C07310=1226.030,289.188,-65.591,-176.498,6.719,148.208
C07311=1226.024,289.461,-65.622,-176.496,6.721,148.208
C07312=1226.020,289.735,-65.655,-176.493,6.724,148.208
C07313=1226.015,290.009,-65.686,-176.491,6.726,148.208
C07314=1226.010,290.258,-65.715,-176.488,6.729,148.208
C07315=1226.006,290.505,-65.743,-176.486,6.731,148.208
C07316=1226.002,290.754,-65.772,-176.483,6.733,148.207
C07317=1225.998,291.003,-65.802,-176.481,6.735,148.207
C07318=1225.994,291.251,-65.830,-176.478,6.738,148.207
C07319=1225.989,291.499,-65.859,-176.476,6.741,148.207
C07320=1225.985,291.748,-65.888,-176.474,6.742,148.207
C07321=1225.980,291.996,-65.917,-176.471,6.746,148.207
C07322=1225.975,292.244,-65.945,-176.469,6.748,148.207
C07323=1225.972,292.492,-65.974,-176.467,6.750,148.207
C07324=1225.967,292.741,-66.003,-176.464,6.752,148.206
C07325=1225.963,292.989,-66.032,-176.462,6.755,148.206
C07326=1225.958,293.237,-66.061,-176.459,6.757,148.206
C07327=1225.954,293.486,-66.090,-176.457,6.759,148.206
C07328=1225.951,293.734,-66.119,-176.455,6.761,148.206
C07329=1225.945,293.982,-66.148,-176.452,6.764,148.206
C07330=1225.941,294.230,-66.177,-176.450,6.767,148.206
C07331=1225.937,294.478,-66.206,-176.448,6.769,148.206
C07332=1225.933,294.727,-66.235,-176.445,6.771,148.206
C07333=1225.928,294.975,-66.265,-176.443,6.774,148.206
C07334=1225.924,295.223,-66.292,-176.440,6.776,148.206
C07335=1225.920,295.472,-66.322,-176.438,6.778,148.206
C07336=1225.916,295.720,-66.351,-176.435,6.781,148.205
C07337=1225.912,295.968,-66.381,-176.433,6.783,148.205
C07338=1225.906,296.216,-66.409,-176.431,6.785,148.205
C07339=1225.902,296.465,-66.439,-176.428,6.788,148.205
C07340=1225.898,296.713,-66.468,-176.426,6.791,148.205
C07341=1225.894,296.962,-66.497,-176.424,6.792,148.205
C07342=1225.889,297.210,-66.526,-176.422,6.795,148.205
C07343=1225.885,297.458,-66.555,-176.419,6.798,148.205
C07344=1225.881,297.706,-66.584,-176.417,6.800,148.205
C07345=1225.877,297.954,-66.614,-176.415,6.802,148.205
C07346=1225.873,298.203,-66.642,-176.412,6.805,148.205
C07347=1225.868,298.451,-66.672,-176.409,6.807,148.204
C07348=1225.864,298.699,-66.701,-176.407,6.809,148.204
C07349=1225.859,298.947,-66.730,-176.405,6.812,148.204
C07350=1225.855,299.195,-66.760,-176.403,6.815,148.204
C07351=1225.851,299.443,-66.789,-176.400,6.817,148.204
C07352=1225.847,299.692,-66.818,-176.398,6.819,148.204
C07353=1225.842,299.941,-66.847,-176.395,6.822,148.204
C07354=1225.838,300.189,-66.877,-176.393,6.824,148.204
C07355=1225.833,300.436,-66.906,-176.391,6.826,148.204
C07356=1225.829,300.685,-66.935,-176.388,6.829,148.204
C07357=1225.825,300.933,-66.965,-176.386,6.831,148.204
C07358=1225.821,301.181,-66.994,-176.384,6.834,148.204
C07359=1225.817,301.429,-67.024,-176.381,6.837,148.204
C07360=1225.812,301.678,-67.054,-176.379,6.839,148.204
C07361=1225.808,301.926,-67.083,-176.377,6.841,148.203
C07362=1225.803,302.175,-67.113,-176.374,6.844,148.203
C07363=1225.799,302.422,-67.142,-176.372,6.846,148.203
C07364=1225.794,302.670,-67.171,-176.370,6.848,148.203
C07365=1225.790,302.919,-67.201,-176.367,6.851,148.203
C07366=1225.786,303.167,-67.230,-176.365,6.854,148.203
C07367=1225.782,303.415,-67.260,-176.363,6.856,148.203
C07368=1225.778,303.663,-67.289,-176.361,6.858,148.203
C07369=1225.774,303.912,-67.319,-176.358,6.861,148.203
C07370=1225.769,304.160,-67.349,-176.356,6.863,148.203
C07371=1225.764,304.409,-67.378,-176.354,6.866,148.203
C07372=1225.760,304.657,-67.408,-176.351,6.868,148.203
C07373=1225.756,304.905,-67.437,-176.349,6.871,148.203
C07374=1225.752,305.153,-67.466,-176.347,6.873,148.203
C07375=1225.748,305.401,-67.497,-176.344,6.876,148.203
C07376=1225.742,305.649,-67.526,-176.342,6.878,148.202
C07377=1225.738,305.897,-67.556,-176.340,6.880,148.202
C07378=1225.734,306.145,-67.585,-176.337,6.883,148.202
C07379=1225.730,306.394,-67.615,-176.335,6.885,148.202
C07380=1225.726,306.642,-67.644,-176.333,6.888,148.202
C07381=1225.721,306.890,-67.675,-176.330,6.891,148.202
C07382=1225.717,307.138,-67.704,-176.328,6.893,148.202
C07383=1225.713,307.386,-67.734,-176.326,6.895,148.202
C07384=1225.709,307.635,-67.763,-176.323,6.898,148.202
C07385=1225.704,307.883,-67.794,-176.321,6.900,148.202
C07386=1225.700,308.131,-67.823,-176.319,6.903,148.202
C07387=1225.696,308.379,-67.853,-176.316,6.906,148.202
C07388=1225.691,308.627,-67.882,-176.314,6.908,148.202
C07389=1225.687,308.875,-67.913,-176.312,6.910,148.202
C07390=1225.683,309.124,-67.943,-176.310,6.913,148.202
C07391=1225.678,309.372,-67.972,-176.307,6.915,148.202
C07392=1225.674,309.620,-68.003,-176.305,6.918,148.202
C07393=1225.670,309.868,-68.032,-176.303,6.921,148.202
C07394=1225.665,310.116,-68.062,-176.301,6.923,148.202
C07395=1225.661,310.364,-68.092,-176.298,6.925,148.202
C07396=1225.657,310.613,-68.122,-176.296,6.928,148.202
C07397=1225.653,310.861,-68.151,-176.294,6.930,148.202
C07398=1225.648,311.109,-68.182,-176.292,6.933,148.202
C07399=1225.644,311.358,-68.212,-176.289,6.936,148.202
C07400=1225.640,311.605,-68.242,-176.287,6.938,148.202
C07401=1225.636,311.854,-68.272,-176.285,6.940,148.202
C07402=1225.631,312.102,-68.302,-176.283,6.944,148.202
C07403=1225.627,312.350,-68.332,-176.280,6.946,148.202
C07404=1225.623,312.599,-68.362,-176.278,6.948,148.202
C07405=1225.619,312.846,-68.392,-176.276,6.951,148.202
C07406=1225.614,313.095,-68.422,-176.274,6.953,148.202
C07407=1225.610,313.342,-68.452,-176.271,6.956,148.202
C07408=1225.606,313.591,-68.482,-176.269,6.958,148.202
C07409=1225.601,313.839,-68.512,-176.267,6.961,148.202
C07410=1225.597,314.087,-68.542,-176.264,6.964,148.202
C07411=1225.592,314.335,-68.573,-176.262,6.966,148.202
C07412=1225.589,314.583,-68.603,-176.260,6.969,148.202
C07413=1225.584,314.832,-68.633,-176.258,6.972,148.202
C07414=1225.579,315.107,-68.667,-176.256,6.974,148.202
C07415=1225.574,315.383,-68.700,-176.253,6.977,148.202
C07416=1225.570,315.658,-68.734,-176.250,6.980,148.202
C07417=1225.565,315.935,-68.767,-176.248,6.982,148.202
C07418=1225.561,316.183,-68.798,-176.246,6.985,148.202
C07419=1225.556,316.431,-68.828,-176.243,6.987,148.202
C07420=1225.553,316.679,-68.858,-176.241,6.991,148.202
C07421=1225.548,316.927,-68.889,-176.239,6.993,148.202
C07422=1225.544,317.176,-68.918,-176.237,6.995,148.202
C07423=1225.540,317.424,-68.949,-176.234,6.998,148.202
C07424=1225.536,317.671,-68.979,-176.232,7.000,148.202
C07425=1225.531,317.920,-69.009,-176.230,7.003,148.202
C07426=1225.526,318.168,-69.040,-176.228,7.006,148.202
C07427=1225.522,318.415,-69.070,-176.226,7.008,148.202
C07428=1225.518,318.664,-69.101,-176.224,7.011,148.202
C07429=1225.514,318.912,-69.131,-176.221,7.014,148.202
C07430=1225.510,319.160,-69.162,-176.219,7.016,148.202
C07431=1225.506,319.408,-69.192,-176.217,7.018,148.202
C07432=1225.501,319.656,-69.223,-176.215,7.021,148.202
C07433=1225.497,319.905,-69.254,-176.213,7.024,148.202
C07434=1225.493,320.153,-69.283,-176.211,7.026,148.202
C07435=1225.488,320.401,-69.314,-176.208,7.029,148.202
C07436=1225.485,320.648,-69.344,-176.206,7.031,148.202
C07437=1225.480,320.896,-69.375,-176.204,7.034,148.202
C07438=1225.476,321.145,-69.406,-176.201,7.037,148.202
C07439=1225.472,321.393,-69.436,-176.200,7.039,148.202
C07440=1225.467,321.641,-69.466,-176.197,7.042,148.202
C07441=1225.462,321.889,-69.497,-176.195,7.044,148.202
C07442=1225.459,322.138,-69.527,-176.193,7.047,148.202
C07443=1225.455,322.386,-69.558,-176.191,7.050,148.202
C07444=1225.450,322.634,-69.589,-176.189,7.052,148.202
C07445=1225.446,322.881,-69.619,-176.187,7.055,148.202
C07446=1225.442,323.130,-69.650,-176.184,7.058,148.202
C07447=1225.437,323.378,-69.681,-176.182,7.060,148.202
C07448=1225.434,323.625,-69.711,-176.180,7.062,148.202
C07449=1225.430,323.874,-69.742,-176.178,7.066,148.202
C07450=1225.425,324.122,-69.773,-176.176,7.068,148.202
C07451=1225.420,324.370,-69.804,-176.173,7.071,148.202
C07452=1225.416,324.618,-69.834,-176.172,7.073,148.203
C07453=1225.412,324.866,-69.865,-176.170,7.076,148.202
C07454=1225.408,325.114,-69.896,-176.167,7.079,148.203
C07455=1225.403,325.362,-69.927,-176.165,7.081,148.203
C07456=1225.400,325.611,-69.957,-176.163,7.084,148.203
C07457=1225.395,325.859,-69.988,-176.160,7.087,148.203
C07458=1225.391,326.107,-70.019,-176.159,7.089,148.203
C07459=1225.387,326.355,-70.050,-176.157,7.091,148.203
C07460=1225.383,326.602,-70.081,-176.155,7.095,148.203
C07461=1225.379,326.850,-70.112,-176.152,7.097,148.203
C07462=1225.375,327.099,-70.143,-176.150,7.099,148.203
C07463=1225.370,327.347,-70.173,-176.148,7.103,148.203
C07464=1225.365,327.595,-70.204,-176.146,7.105,148.203
C07465=1225.361,327.843,-70.235,-176.144,7.108,148.203
C07466=1225.357,328.091,-70.266,-176.142,7.110,148.203
C07467=1225.353,328.338,-70.297,-176.140,7.113,148.203
C07468=1225.349,328.587,-70.328,-176.138,7.116,148.203
C07469=1225.344,328.835,-70.359,-176.135,7.118,148.203
C07470=1225.340,329.083,-70.390,-176.134,7.121,148.204
C07471=1225.336,329.332,-70.421,-176.131,7.124,148.204
C07472=1225.332,329.579,-70.452,-176.130,7.126,148.204
C07473=1225.327,329.827,-70.483,-176.127,7.128,148.204
C07474=1225.324,330.075,-70.514,-176.125,7.132,148.204
C07475=1225.319,330.323,-70.544,-176.123,7.134,148.204
C07476=1225.315,330.571,-70.576,-176.121,7.137,148.204
C07477=1225.311,330.819,-70.607,-176.119,7.140,148.204
C07478=1225.306,331.067,-70.638,-176.117,7.142,148.204
C07479=1225.302,331.315,-70.670,-176.115,7.144,148.204
C07480=1225.298,331.563,-70.700,-176.113,7.148,148.204
C07481=1225.294,331.812,-70.731,-176.111,7.150,148.204
C07482=1225.289,332.059,-70.763,-176.109,7.152,148.205
C07483=1225.285,332.307,-70.794,-176.107,7.156,148.205
C07484=1225.281,332.556,-70.825,-176.105,7.158,148.205
C07485=1225.277,332.803,-70.856,-176.102,7.161,148.205
C07486=1225.273,333.052,-70.887,-176.101,7.164,148.205
C07487=1225.268,333.299,-70.919,-176.099,7.166,148.205
C07488=1225.264,333.548,-70.950,-176.096,7.169,148.205
C07489=1225.260,333.796,-70.981,-176.094,7.171,148.205
C07490=1225.256,334.044,-71.013,-176.093,7.174,148.205
C07491=1225.251,334.292,-71.043,-176.090,7.177,148.206
C07492=1225.247,334.539,-71.075,-176.088,7.180,148.205
C07493=1225.243,334.788,-71.106,-176.087,7.182,148.206
C07494=1225.239,335.035,-71.137,-176.084,7.185,148.206
C07495=1225.235,335.284,-71.169,-176.082,7.188,148.206
C07496=1225.230,335.531,-71.200,-176.081,7.190,148.206
C07497=1225.226,335.780,-71.231,-176.078,7.193,148.206
C07498=1225.222,336.027,-71.263,-176.077,7.196,148.206
C07499=1225.218,336.276,-71.294,-176.074,7.198,148.206
C07500=1225.214,336.523,-71.325,-176.072,7.201,148.206
C07501=1225.210,336.772,-71.356,-176.071,7.204,148.207
C07502=1225.205,337.019,-71.389,-176.069,7.206,148.207
C07503=1225.201,337.267,-71.420,-176.066,7.210,148.207
C07504=1225.196,337.515,-71.451,-176.065,7.212,148.207
C07505=1225.193,337.763,-71.483,-176.063,7.214,148.207
C07506=1225.188,338.011,-71.514,-176.060,7.218,148.207
C07507=1225.184,338.259,-71.546,-176.059,7.220,148.207
C07508=1225.180,338.507,-71.577,-176.057,7.222,148.207
C07509=1225.176,338.755,-71.608,-176.055,7.226,148.208
C07510=1225.171,339.003,-71.640,-176.053,7.228,148.208
C07511=1225.167,339.251,-71.672,-176.051,7.231,148.208
C07512=1225.163,339.500,-71.703,-176.049,7.234,148.208
C07513=1225.159,339.747,-71.735,-176.047,7.236,148.208
C07514=1225.155,339.995,-71.767,-176.045,7.239,148.208
C07515=1225.151,340.243,-71.797,-176.043,7.242,148.208
C07516=1225.146,340.491,-71.830,-176.041,7.245,148.208
C07517=1225.142,340.739,-71.861,-176.039,7.247,148.209
C07518=1225.137,341.017,-71.896,-176.037,7.250,148.209
C07519=1225.133,341.294,-71.932,-176.035,7.253,148.209
C07520=1225.128,341.572,-71.968,-176.033,7.256,148.209
C07521=1225.123,341.850,-72.003,-176.031,7.259,148.209
C07522=1225.119,342.098,-72.034,-176.029,7.263,148.210
C07523=1225.115,342.346,-72.066,-176.027,7.265,148.209
C07524=1225.110,342.593,-72.098,-176.025,7.267,148.210
C07525=1225.106,342.842,-72.130,-176.023,7.270,148.210
C07526=1225.103,343.090,-72.162,-176.021,7.273,148.210
C07527=1225.098,343.338,-72.193,-176.019,7.276,148.210
C07528=1225.094,343.586,-72.225,-176.017,7.278,148.210
C07529=1225.089,343.833,-72.257,-176.015,7.281,148.210
C07530=1225.086,344.081,-72.288,-176.014,7.284,148.211
C07531=1225.081,344.330,-72.321,-176.012,7.287,148.211
C07532=1225.077,344.577,-72.352,-176.010,7.290,148.211
C07533=1225.073,344.825,-72.384,-176.008,7.292,148.211
C07534=1225.068,345.073,-72.416,-176.006,7.295,148.211
C07535=1225.064,345.321,-72.448,-176.004,7.298,148.211
C07536=1225.060,345.569,-72.479,-176.002,7.301,148.212
C07537=1225.055,345.817,-72.511,-176.001,7.303,148.212
C07538=1225.052,346.065,-72.543,-175.999,7.306,148.212
C07539=1225.048,346.313,-72.575,-175.997,7.309,148.212
C07540=1225.043,346.561,-72.607,-175.995,7.311,148.212
C07541=1225.039,346.809,-72.639,-175.993,7.314,148.213
C07542=1225.036,347.057,-72.671,-175.991,7.317,148.213
C07543=1225.030,347.304,-72.703,-175.990,7.320,148.213
C07544=1225.027,347.552,-72.735,-175.988,7.322,148.213
C07545=1225.022,347.801,-72.767,-175.986,7.326,148.213
C07546=1225.018,348.048,-72.799,-175.984,7.328,148.214
C07547=1225.015,348.296,-72.831,-175.983,7.331,148.214
C07548=1225.010,348.544,-72.864,-175.980,7.333,148.214
C07549=1225.006,348.791,-72.895,-175.978,7.336,148.214
C07550=1225.001,349.040,-72.928,-175.977,7.339,148.214
C07551=1224.998,349.288,-72.959,-175.975,7.341,148.214
C07552=1224.993,349.535,-72.991,-175.973,7.345,148.215
C07553=1224.989,349.783,-73.023,-175.971,7.347,148.215
C07554=1224.985,350.032,-73.056,-175.970,7.350,148.215
C07555=1224.981,350.280,-73.088,-175.968,7.352,148.215
C07556=1224.976,350.527,-73.120,-175.966,7.356,148.216
C07557=1224.972,350.775,-73.152,-175.965,7.359,148.216
C07558=1224.969,351.023,-73.184,-175.963,7.361,148.216
C07559=1224.964,351.270,-73.216,-175.961,7.364,148.216
C07560=1224.960,351.518,-73.248,-175.959,7.367,148.216
C07561=1224.955,351.767,-73.280,-175.958,7.370,148.216
C07562=1224.952,352.014,-73.313,-175.956,7.372,148.217
C07563=1224.947,352.262,-73.345,-175.954,7.375,148.217
C07564=1224.943,352.510,-73.378,-175.952,7.378,148.217
C07565=1224.939,352.758,-73.409,-175.950,7.381,148.217
C07566=1224.935,353.006,-73.443,-175.949,7.383,148.217
C07567=1224.930,353.253,-73.474,-175.947,7.386,148.218
C07568=1224.926,353.502,-73.506,-175.945,7.389,148.218
C07569=1224.922,353.750,-73.538,-175.944,7.392,148.218
C07570=1224.918,353.997,-73.571,-175.942,7.394,148.218
C07571=1224.914,354.245,-73.603,-175.940,7.398,148.219
C07572=1224.909,354.493,-73.635,-175.938,7.400,148.219
C07573=1224.905,354.741,-73.669,-175.937,7.403,148.219
C07574=1224.902,354.989,-73.700,-175.935,7.405,148.219
C07575=1224.897,355.237,-73.733,-175.934,7.408,148.220
C07576=1224.893,355.484,-73.765,-175.932,7.411,148.220
C07577=1224.889,355.732,-73.797,-175.930,7.414,148.220
C07578=1224.885,355.980,-73.831,-175.929,7.416,148.220
C07579=1224.881,356.228,-73.862,-175.927,7.419,148.220
C07580=1224.876,356.476,-73.895,-175.925,7.423,148.221
C07581=1224.872,356.723,-73.927,-175.924,7.425,148.221
C07582=1224.868,356.972,-73.960,-175.922,7.428,148.221
C07583=1224.864,357.219,-73.993,-175.920,7.430,148.221
C07584=1224.860,357.467,-74.025,-175.918,7.434,148.222
C07585=1224.856,357.715,-74.058,-175.917,7.436,148.222
C07586=1224.851,357.963,-74.090,-175.915,7.439,148.222
C07587=1224.847,358.211,-74.122,-175.914,7.441,148.222
C07588=1224.843,358.458,-74.155,-175.913,7.444,148.223
C07589=1224.839,358.707,-74.187,-175.910,7.448,148.223
C07590=1224.835,358.954,-74.220,-175.909,7.450,148.223
C07591=1224.831,359.203,-74.252,-175.907,7.453,148.223
C07592=1224.827,359.450,-74.285,-175.906,7.456,148.224
C07593=1224.822,359.699,-74.318,-175.904,7.458,148.224
C07594=1224.818,359.945,-74.350,-175.902,7.461,148.224
C07595=1224.814,360.193,-74.383,-175.901,7.464,148.225
C07596=1224.810,360.441,-74.416,-175.899,7.467,148.225
C07597=1224.806,360.689,-74.448,-175.898,7.469,148.225
C07598=1224.802,360.937,-74.481,-175.896,7.472,148.225
C07599=1224.798,361.185,-74.514,-175.894,7.475,148.226
C07600=1224.793,361.433,-74.547,-175.893,7.478,148.226
C07601=1224.790,361.681,-74.579,-175.891,7.481,148.226
C07602=1224.786,361.928,-74.612,-175.890,7.483,148.226
C07603=1224.781,362.176,-74.644,-175.889,7.486,148.227
C07604=1224.776,362.424,-74.677,-175.887,7.489,148.227
C07605=1224.772,362.672,-74.710,-175.885,7.492,148.227
C07606=1224.769,362.920,-74.742,-175.884,7.495,148.228
C07607=1224.764,363.167,-74.775,-175.882,7.497,148.228
C07608=1224.760,363.415,-74.808,-175.881,7.500,148.228
C07609=1224.756,363.663,-74.841,-175.879,7.503,148.228
C07610=1224.752,363.911,-74.874,-175.878,7.506,148.229
C07611=1224.748,364.159,-74.907,-175.876,7.508,148.229
C07612=1224.744,364.406,-74.940,-175.875,7.512,148.229
C07613=1224.740,364.655,-74.972,-175.873,7.514,148.230
C07614=1224.736,364.902,-75.005,-175.872,7.517,148.230
C07615=1224.731,365.150,-75.039,-175.870,7.520,148.230
C07616=1224.728,365.397,-75.071,-175.869,7.522,148.231
C07617=1224.723,365.645,-75.103,-175.868,7.525,148.231
C07618=1224.719,365.893,-75.136,-175.866,7.528,148.231
C07619=1224.715,366.141,-75.169,-175.865,7.530,148.231
C07620=1224.711,366.388,-75.203,-175.864,7.533,148.232
C07621=1224.706,366.637,-75.235,-175.861,7.537,148.232
C07622=1224.702,366.916,-75.273,-175.860,7.539,148.232
C07623=1224.697,367.196,-75.310,-175.858,7.543,148.233
C07624=1224.693,367.476,-75.346,-175.857,7.546,148.233
C07625=1224.688,367.755,-75.384,-175.855,7.549,148.233
C07626=1224.684,368.003,-75.417,-175.854,7.552,148.234
C07627=1224.680,368.251,-75.450,-175.852,7.555,148.234
C07628=1224.676,368.499,-75.483,-175.851,7.557,148.234
C07629=1224.672,368.746,-75.516,-175.850,7.560,148.235
C07630=1224.668,368.994,-75.550,-175.848,7.563,148.235
C07631=1224.663,369.242,-75.582,-175.847,7.566,148.235
C07632=1224.659,369.490,-75.615,-175.846,7.568,148.236
C07633=1224.655,369.738,-75.648,-175.844,7.571,148.236
C07634=1224.651,369.986,-75.682,-175.843,7.574,148.236
C07635=1224.647,370.233,-75.715,-175.842,7.577,148.237
C07636=1224.642,370.481,-75.748,-175.840,7.579,148.237
C07637=1224.638,370.729,-75.781,-175.839,7.582,148.237
C07638=1224.634,370.976,-75.814,-175.838,7.585,148.238
C07639=1224.630,371.224,-75.847,-175.836,7.587,148.238
C07640=1224.626,371.472,-75.880,-175.835,7.590,148.238
C07641=1224.622,371.720,-75.914,-175.834,7.593,148.239
C07642=1224.618,371.967,-75.947,-175.833,7.596,148.239
C07643=1224.613,372.215,-75.980,-175.831,7.598,148.239
C07644=1224.609,372.463,-76.013,-175.830,7.601,148.240
C07645=1224.605,372.711,-76.046,-175.829,7.604,148.240
C07646=1224.601,372.958,-76.079,-175.828,7.607,148.241
C07647=1224.597,373.206,-76.113,-175.826,7.609,148.241
C07648=1224.593,373.454,-76.146,-175.825,7.612,148.241
C07649=1224.589,373.702,-76.179,-175.824,7.615,148.242
C07650=1224.585,373.950,-76.212,-175.823,7.618,148.242
C07651=1224.581,374.198,-76.246,-175.821,7.621,148.242
C07652=1224.577,374.445,-76.279,-175.820,7.623,148.242
C07653=1224.573,374.692,-76.313,-175.819,7.626,148.243
C07654=1224.569,374.940,-76.346,-175.817,7.629,148.243
C07655=1224.565,375.188,-76.379,-175.816,7.632,148.244
C07656=1224.560,375.436,-76.413,-175.815,7.634,148.244
C07657=1224.556,375.684,-76.446,-175.814,7.637,148.244
C07658=1224.552,375.931,-76.479,-175.813,7.639,148.245
C07659=1224.547,376.179,-76.512,-175.812,7.642,148.245
C07660=1224.544,376.426,-76.546,-175.810,7.644,148.245
C07661=1224.540,376.675,-76.580,-175.809,7.647,148.246
C07662=1224.536,376.922,-76.613,-175.808,7.650,148.246
C07663=1224.532,377.170,-76.646,-175.807,7.653,148.247
C07664=1224.528,377.418,-76.679,-175.806,7.656,148.247
C07665=1224.523,377.666,-76.713,-175.805,7.659,148.247
C07666=1224.519,377.913,-76.747,-175.803,7.661,148.248
C07667=1224.515,378.161,-76.780,-175.803,7.663,148.248
C07668=1224.511,378.408,-76.813,-175.802,7.666,148.249
C07669=1224.506,378.656,-76.846,-175.800,7.669,148.249
C07670=1224.503,378.904,-76.880,-175.799,7.672,148.249
C07671=1224.498,379.152,-76.914,-175.798,7.675,148.250
C07672=1224.494,379.400,-76.947,-175.796,7.677,148.250
C07673=1224.490,379.648,-76.980,-175.796,7.679,148.250
C07674=1224.486,379.895,-77.014,-175.795,7.682,148.251
C07675=1224.482,380.142,-77.047,-175.793,7.685,148.251
C07676=1224.478,380.390,-77.081,-175.792,7.688,148.251
C07677=1224.474,380.638,-77.115,-175.791,7.690,148.252
C07678=1224.470,380.886,-77.149,-175.790,7.693,148.252
C07679=1224.466,381.134,-77.182,-175.789,7.695,148.253
C07680=1224.462,381.381,-77.216,-175.789,7.698,148.253
C07681=1224.457,381.629,-77.249,-175.787,7.701,148.254
C07682=1224.453,381.877,-77.282,-175.786,7.704,148.254
C07683=1224.449,382.124,-77.316,-175.785,7.707,148.254
C07684=1224.446,382.372,-77.350,-175.784,7.709,148.255
C07685=1224.441,382.620,-77.383,-175.783,7.712,148.255
C07686=1224.437,382.867,-77.417,-175.782,7.714,148.256
C07687=1224.433,383.115,-77.451,-175.781,7.717,148.256
C07688=1224.429,383.363,-77.484,-175.780,7.719,148.256
C07689=1224.425,383.611,-77.519,-175.779,7.722,148.257
C07690=1224.420,383.859,-77.552,-175.778,7.725,148.257
C07691=1224.417,384.106,-77.586,-175.777,7.728,148.257
C07692=1224.412,384.353,-77.619,-175.776,7.730,148.258
C07693=1224.408,384.601,-77.653,-175.775,7.733,148.258
C07694=1224.404,384.849,-77.686,-175.774,7.736,148.259
C07695=1224.400,385.097,-77.720,-175.774,7.738,148.259
C07696=1224.396,385.344,-77.754,-175.772,7.740,148.260
C07697=1224.392,385.592,-77.788,-175.771,7.743,148.260
C07698=1224.388,385.839,-77.821,-175.770,7.746,148.260
C07699=1224.384,386.087,-77.855,-175.769,7.748,148.261
C07700=1224.380,386.335,-77.889,-175.768,7.751,148.261
C07701=1224.375,386.583,-77.923,-175.767,7.754,148.261
C07702=1224.372,386.830,-77.956,-175.767,7.756,148.262
C07703=1224.367,387.078,-77.990,-175.766,7.759,148.262
C07704=1224.364,387.326,-78.024,-175.765,7.762,148.263
C07705=1224.359,387.573,-78.058,-175.764,7.764,148.263
C07706=1224.355,387.821,-78.092,-175.763,7.766,148.264
C07707=1224.351,388.069,-78.125,-175.762,7.769,148.264
C07708=1224.347,388.316,-78.159,-175.761,7.772,148.264
C07709=1224.343,388.564,-78.193,-175.760,7.774,148.265
C07710=1224.339,388.812,-78.227,-175.759,7.777,148.265
C07711=1224.334,389.059,-78.262,-175.758,7.779,148.266
C07712=1224.331,389.307,-78.295,-175.757,7.782,148.266
C07713=1224.327,389.555,-78.329,-175.757,7.784,148.267
C07714=1224.322,389.803,-78.363,-175.756,7.787,148.267
C07715=1224.318,390.050,-78.397,-175.755,7.790,148.267
C07716=1224.315,390.297,-78.431,-175.754,7.792,148.268
C07717=1224.310,390.546,-78.465,-175.753,7.795,148.268
C07718=1224.306,390.793,-78.498,-175.753,7.797,148.269
C07719=1224.301,391.041,-78.532,-175.752,7.800,148.269
C07720=1224.298,391.288,-78.566,-175.750,7.803,148.269
C07721=1224.294,391.536,-78.600,-175.750,7.805,148.270
C07722=1224.289,391.784,-78.634,-175.749,7.808,148.270
C07723=1224.285,392.031,-78.668,-175.748,7.810,148.271
C07724=1224.282,392.279,-78.703,-175.747,7.812,148.271
C07725=1224.277,392.527,-78.736,-175.747,7.814,148.271
C07726=1224.273,392.808,-78.775,-175.746,7.818,148.272
C07727=1224.268,393.090,-78.813,-175.745,7.820,148.272
C07728=1224.264,393.372,-78.852,-175.744,7.824,148.273
C07729=1224.258,393.652,-78.891,-175.743,7.826,148.273
C07730=1224.255,393.901,-78.925,-175.742,7.828,148.274
C07731=1224.251,394.148,-78.959,-175.741,7.831,148.274
C07732=1224.247,394.395,-78.993,-175.741,7.833,148.275
C07733=1224.243,394.644,-79.027,-175.740,7.836,148.275
C07734=1224.238,394.891,-79.061,-175.739,7.838,148.275
C07735=1224.235,395.138,-79.095,-175.738,7.841,148.276
C07736=1224.231,395.386,-79.130,-175.738,7.843,148.276
C07737=1224.226,395.634,-79.163,-175.736,7.846,148.277
C07738=1224.222,395.882,-79.198,-175.736,7.848,148.277
C07739=1224.218,396.129,-79.231,-175.735,7.851,148.278
C07740=1224.214,396.377,-79.266,-175.734,7.853,148.278
C07741=1224.210,396.624,-79.300,-175.734,7.856,148.279
C07742=1224.205,396.872,-79.334,-175.733,7.858,148.279
C07743=1224.202,397.120,-79.368,-175.732,7.860,148.279
C07744=1224.198,397.367,-79.403,-175.731,7.863,148.280
C07745=1224.194,397.614,-79.437,-175.731,7.865,148.280
C07746=1224.190,397.862,-79.471,-175.730,7.868,148.281
C07747=1224.186,398.110,-79.505,-175.729,7.870,148.281
C07748=1224.181,398.358,-79.539,-175.729,7.873,148.282
C07749=1224.177,398.606,-79.574,-175.728,7.875,148.282
C07750=1224.173,398.853,-79.608,-175.727,7.877,148.282
C07751=1224.169,399.100,-79.642,-175.727,7.880,148.283
C07752=1224.165,399.348,-79.676,-175.726,7.882,148.283
C07753=1224.161,399.595,-79.711,-175.725,7.885,148.284
C07754=1224.157,399.844,-79.744,-175.725,7.887,148.284
C07755=1224.153,400.091,-79.779,-175.724,7.889,148.285
C07756=1224.149,400.338,-79.813,-175.723,7.892,148.285
C07757=1224.145,400.587,-79.848,-175.723,7.894,148.286
C07758=1224.140,400.834,-79.882,-175.722,7.896,148.286
C07759=1224.137,401.081,-79.916,-175.721,7.899,148.286
C07760=1224.133,401.329,-79.951,-175.721,7.902,148.287
C07761=1224.129,401.576,-79.985,-175.720,7.904,148.287
C07762=1224.124,401.824,-80.019,-175.719,7.907,148.288
C07763=1224.120,402.072,-80.054,-175.719,7.909,148.288
C07764=1224.116,402.320,-80.087,-175.718,7.911,148.288
C07765=1224.112,402.568,-80.122,-175.717,7.914,148.289
C07766=1224.108,402.815,-80.156,-175.717,7.916,148.289
C07767=1224.104,403.062,-80.190,-175.716,7.918,148.290
C07768=1224.100,403.310,-80.225,-175.715,7.921,148.290
C07769=1224.096,403.557,-80.259,-175.715,7.923,148.291
C07770=1224.092,403.806,-80.294,-175.714,7.925,148.291
C07771=1224.087,404.053,-80.328,-175.713,7.928,148.292
C07772=1224.084,404.300,-80.362,-175.713,7.930,148.292
C07773=1224.080,404.548,-80.397,-175.712,7.932,148.292
C07774=1224.076,404.795,-80.431,-175.712,7.934,148.293
C07775=1224.072,405.043,-80.466,-175.711,7.937,148.293
C07776=1224.067,405.291,-80.500,-175.710,7.939,148.294
C07777=1224.063,405.538,-80.534,-175.710,7.941,148.294
C07778=1224.059,405.786,-80.569,-175.709,7.944,148.295
C07779=1224.055,406.034,-80.603,-175.708,7.946,148.295
C07780=1224.052,406.281,-80.637,-175.708,7.948,148.295
C07781=1224.047,406.529,-80.672,-175.707,7.950,148.296
C07782=1224.042,406.776,-80.706,-175.706,7.953,148.296
C07783=1224.040,407.023,-80.741,-175.706,7.955,148.297
C07784=1224.035,407.271,-80.776,-175.706,7.958,148.297
C07785=1224.031,407.519,-80.811,-175.705,7.960,148.298
C07786=1224.027,407.766,-80.845,-175.704,7.961,148.298
C07787=1224.023,408.014,-80.879,-175.704,7.965,148.298
C07788=1224.019,408.262,-80.914,-175.703,7.967,148.299
C07789=1224.015,408.509,-80.948,-175.702,7.969,148.299
C07790=1224.011,408.757,-80.983,-175.702,7.971,148.300
C07791=1224.006,409.004,-81.017,-175.701,7.973,148.300
C07792=1224.002,409.252,-81.052,-175.701,7.976,148.301
C07793=1223.998,409.499,-81.086,-175.700,7.978,148.301
C07794=1223.995,409.747,-81.121,-175.699,7.980,148.301
C07795=1223.990,409.994,-81.156,-175.699,7.982,148.302
C07796=1223.987,410.242,-81.190,-175.699,7.984,148.302
C07797=1223.982,410.490,-81.224,-175.697,7.987,148.303
C07798=1223.978,410.737,-81.259,-175.697,7.989,148.303
C07799=1223.974,410.985,-81.294,-175.697,7.991,148.303
C07800=1223.970,411.232,-81.328,-175.696,7.993,148.304
C07801=1223.966,411.480,-81.363,-175.696,7.995,148.304
C07802=1223.962,411.727,-81.398,-175.695,7.997,148.305
C07803=1223.958,411.975,-81.432,-175.694,8.001,148.305
C07804=1223.954,412.222,-81.466,-175.694,8.003,148.306
C07805=1223.950,412.471,-81.501,-175.693,8.004,148.306
C07806=1223.946,412.718,-81.536,-175.693,8.007,148.307
C07807=1223.942,412.965,-81.571,-175.692,8.009,148.307
C07808=1223.938,413.213,-81.605,-175.692,8.011,148.307
C07809=1223.934,413.461,-81.640,-175.691,8.013,148.308
C07810=1223.929,413.708,-81.674,-175.691,8.015,148.308
C07811=1223.926,413.956,-81.710,-175.690,8.018,148.309
C07812=1223.922,414.203,-81.744,-175.689,8.020,148.309
C07813=1223.918,414.451,-81.779,-175.689,8.022,148.309
C07814=1223.913,414.698,-81.813,-175.689,8.024,148.310
C07815=1223.909,414.946,-81.848,-175.688,8.026,148.310
C07816=1223.905,415.193,-81.883,-175.687,8.028,148.311
C07817=1223.902,415.441,-81.917,-175.687,8.031,148.311
C07818=1223.894,415.853,-81.975,-175.686,8.034,148.312
C07819=1223.888,416.266,-82.033,-175.685,8.038,148.312
C07820=1223.881,416.679,-82.091,-175.684,8.042,148.313
C07821=1223.877,417.092,-82.149,-175.684,8.045,148.314
C07822=1223.456,417.092,-82.183,-175.687,8.055,148.317
C07823=1223.459,416.676,-82.125,-175.687,8.052,148.317
C07824=1223.466,416.261,-82.066,-175.689,8.048,148.316
C07825=1223.473,415.845,-82.008,-175.689,8.045,148.315
C07826=1223.480,415.430,-81.950,-175.690,8.041,148.315
C07827=1223.484,415.183,-81.915,-175.691,8.039,148.314
C07828=1223.487,414.935,-81.880,-175.691,8.037,148.314
C07829=1223.492,414.688,-81.846,-175.692,8.035,148.313
C07830=1223.496,414.440,-81.811,-175.692,8.033,148.313
C07831=1223.500,414.192,-81.776,-175.692,8.030,148.313
C07832=1223.504,413.945,-81.741,-175.694,8.028,148.312
C07833=1223.508,413.698,-81.707,-175.694,8.026,148.312
C07834=1223.512,413.450,-81.672,-175.694,8.023,148.311
C07835=1223.516,413.202,-81.638,-175.695,8.021,148.311
C07836=1223.520,412.954,-81.603,-175.696,8.019,148.311
C07837=1223.524,412.708,-81.568,-175.696,8.017,148.310
C07838=1223.528,412.460,-81.533,-175.697,8.015,148.310
C07839=1223.532,412.212,-81.499,-175.697,8.013,148.309
C07840=1223.536,411.964,-81.464,-175.698,8.010,148.309
C07841=1223.540,411.717,-81.430,-175.699,8.008,148.308
C07842=1223.544,411.469,-81.395,-175.699,8.006,148.308
C07843=1223.548,411.222,-81.360,-175.699,8.004,148.308
C07844=1223.552,410.974,-81.325,-175.700,8.002,148.307
C07845=1223.556,410.727,-81.292,-175.700,8.000,148.307
C07846=1223.561,410.479,-81.257,-175.701,7.998,148.306
C07847=1223.565,410.231,-81.222,-175.702,7.994,148.306
C07848=1223.569,409.984,-81.187,-175.702,7.992,148.305
C07849=1223.572,409.737,-81.153,-175.703,7.991,148.305
C07850=1223.577,409.489,-81.118,-175.703,7.988,148.305
C07851=1223.581,409.241,-81.084,-175.704,7.986,148.304
C07852=1223.584,408.994,-81.050,-175.704,7.983,148.304
C07853=1223.588,408.746,-81.015,-175.705,7.981,148.303
C07854=1223.593,408.498,-80.980,-175.706,7.979,148.303
C07855=1223.597,408.250,-80.946,-175.706,7.977,148.302
C07856=1223.601,408.004,-80.911,-175.707,7.975,148.302
C07857=1223.605,407.756,-80.876,-175.708,7.972,148.302
C07858=1223.609,407.508,-80.842,-175.708,7.970,148.301
C07859=1223.613,407.261,-80.808,-175.709,7.968,148.301
C07860=1223.617,407.013,-80.773,-175.709,7.966,148.300
C07861=1223.621,406.766,-80.738,-175.709,7.964,148.300
C07862=1223.625,406.518,-80.704,-175.711,7.961,148.300
C07863=1223.629,406.270,-80.670,-175.711,7.959,148.299
C07864=1223.634,406.023,-80.635,-175.711,7.957,148.299
C07865=1223.637,405.775,-80.601,-175.712,7.955,148.298
C07866=1223.642,405.528,-80.567,-175.713,7.951,148.298
C07867=1223.646,405.280,-80.532,-175.713,7.949,148.297
C07868=1223.649,405.033,-80.498,-175.714,7.947,148.297
C07869=1223.654,404.785,-80.463,-175.715,7.944,148.296
C07870=1223.658,404.537,-80.429,-175.715,7.942,148.296
C07871=1223.662,404.290,-80.395,-175.716,7.940,148.296
C07872=1223.666,404.042,-80.360,-175.716,7.938,148.295
C07873=1223.670,403.794,-80.325,-175.717,7.935,148.295
C07874=1223.674,403.547,-80.292,-175.718,7.933,148.294
C07875=1223.678,403.299,-80.257,-175.718,7.931,148.294
C07876=1223.682,403.052,-80.223,-175.719,7.928,148.293
C07877=1223.686,402.804,-80.188,-175.720,7.926,148.293
C07878=1223.690,402.556,-80.154,-175.720,7.924,148.293
C07879=1223.694,402.309,-80.120,-175.721,7.921,148.292
C07880=1223.698,402.061,-80.085,-175.722,7.919,148.292
C07881=1223.703,401.814,-80.050,-175.722,7.917,148.291
C07882=1223.706,401.566,-80.016,-175.723,7.914,148.291
C07883=1223.711,401.319,-79.982,-175.724,7.912,148.290
C07884=1223.714,401.072,-79.948,-175.724,7.910,148.290
C07885=1223.718,400.823,-79.913,-175.725,7.907,148.289
C07886=1223.722,400.576,-79.879,-175.726,7.905,148.289
C07887=1223.727,400.328,-79.845,-175.726,7.903,148.289
C07888=1223.731,400.080,-79.811,-175.727,7.900,148.288
C07889=1223.735,399.833,-79.777,-175.728,7.898,148.288
C07890=1223.739,399.585,-79.742,-175.728,7.895,148.287
C07891=1223.743,399.338,-79.708,-175.729,7.893,148.287
C07892=1223.747,399.090,-79.673,-175.730,7.891,148.287
C07893=1223.751,398.843,-79.639,-175.730,7.888,148.286
C07894=1223.755,398.595,-79.605,-175.731,7.886,148.286
C07895=1223.760,398.347,-79.571,-175.732,7.884,148.285
C07896=1223.763,398.099,-79.537,-175.732,7.880,148.285
C07897=1223.768,397.852,-79.502,-175.733,7.879,148.284
C07898=1223.772,397.605,-79.468,-175.734,7.876,148.284
C07899=1223.776,397.357,-79.434,-175.734,7.873,148.283
C07900=1223.779,397.110,-79.400,-175.735,7.871,148.283
C07901=1223.784,396.861,-79.366,-175.736,7.869,148.283
C07902=1223.788,396.614,-79.332,-175.736,7.866,148.282
C07903=1223.792,396.366,-79.297,-175.737,7.864,148.282
C07904=1223.796,396.119,-79.263,-175.738,7.862,148.281
C07905=1223.800,395.871,-79.229,-175.739,7.858,148.281
C07906=1223.804,395.623,-79.195,-175.739,7.856,148.280
C07907=1223.809,395.376,-79.161,-175.741,7.854,148.280
C07908=1223.812,395.128,-79.127,-175.741,7.852,148.280
C07909=1223.816,394.881,-79.092,-175.742,7.849,148.279
C07910=1223.821,394.633,-79.059,-175.743,7.847,148.279
C07911=1223.825,394.386,-79.025,-175.744,7.844,148.278
C07912=1223.828,394.138,-78.990,-175.744,7.841,148.278
C07913=1223.833,393.890,-78.956,-175.745,7.839,148.277
C07914=1223.837,393.643,-78.923,-175.746,7.837,148.277
C07915=1223.842,393.361,-78.883,-175.747,7.834,148.276
C07916=1223.846,393.079,-78.845,-175.748,7.831,148.276
C07917=1223.851,392.798,-78.806,-175.748,7.828,148.275
C07918=1223.855,392.516,-78.767,-175.750,7.825,148.275
C07919=1223.860,392.268,-78.734,-175.750,7.823,148.275
C07920=1223.863,392.021,-78.700,-175.751,7.820,148.274
C07921=1223.867,391.773,-78.665,-175.752,7.818,148.274
C07922=1223.871,391.525,-78.632,-175.753,7.815,148.273
C07923=1223.876,391.278,-78.597,-175.753,7.813,148.273
C07924=1223.879,391.030,-78.563,-175.755,7.810,148.273
C07925=1223.884,390.782,-78.529,-175.755,7.807,148.272
C07926=1223.888,390.535,-78.496,-175.756,7.805,148.272
C07927=1223.892,390.287,-78.462,-175.757,7.802,148.271
C07928=1223.896,390.039,-78.428,-175.758,7.800,148.271
C07929=1223.900,389.792,-78.394,-175.759,7.797,148.270
C07930=1223.905,389.544,-78.360,-175.760,7.794,148.270
C07931=1223.909,389.297,-78.326,-175.760,7.792,148.270
C07932=1223.912,389.048,-78.293,-175.762,7.790,148.269
C07933=1223.917,388.801,-78.258,-175.762,7.788,148.269
C07934=1223.921,388.554,-78.224,-175.763,7.784,148.268
C07935=1223.925,388.306,-78.191,-175.764,7.782,148.268
C07936=1223.929,388.058,-78.156,-175.765,7.780,148.268
C07937=1223.933,387.810,-78.123,-175.766,7.777,148.267
C07938=1223.937,387.563,-78.089,-175.767,7.774,148.267
C07939=1223.942,387.315,-78.055,-175.767,7.772,148.266
C07940=1223.945,387.067,-78.021,-175.768,7.769,148.266
C07941=1223.950,386.819,-77.987,-175.770,7.766,148.265
C07942=1223.953,386.572,-77.954,-175.770,7.764,148.265
C07943=1223.958,386.324,-77.920,-175.771,7.761,148.265
C07944=1223.962,386.077,-77.886,-175.773,7.758,148.264
C07945=1223.966,385.829,-77.852,-175.773,7.756,148.264
C07946=1223.970,385.581,-77.819,-175.774,7.753,148.263
C07947=1223.974,385.334,-77.785,-175.775,7.751,148.263
C07948=1223.978,385.086,-77.751,-175.776,7.748,148.263
C07949=1223.982,384.838,-77.717,-175.777,7.746,148.262
C07950=1223.986,384.591,-77.684,-175.778,7.743,148.262
C07951=1223.991,384.343,-77.650,-175.779,7.740,148.261
C07952=1223.994,384.096,-77.616,-175.780,7.738,148.261
C07953=1223.998,383.848,-77.583,-175.781,7.735,148.261
C07954=1224.003,383.600,-77.550,-175.782,7.732,148.260
C07955=1224.007,383.352,-77.515,-175.783,7.729,148.260
C07956=1224.011,383.104,-77.482,-175.784,7.727,148.259
C07957=1224.015,382.857,-77.448,-175.785,7.725,148.259
C07958=1224.019,382.609,-77.414,-175.786,7.722,148.259
C07959=1224.024,382.361,-77.381,-175.787,7.719,148.258
C07960=1224.027,382.114,-77.347,-175.788,7.716,148.258
C07961=1224.031,381.866,-77.313,-175.789,7.714,148.257
C07962=1224.036,381.619,-77.279,-175.790,7.711,148.257
C07963=1224.040,381.371,-77.246,-175.791,7.708,148.257
C07964=1224.044,381.123,-77.213,-175.792,7.706,148.256
C07965=1224.048,380.876,-77.179,-175.794,7.703,148.256
C07966=1224.051,380.628,-77.145,-175.794,7.701,148.255
C07967=1224.056,380.379,-77.112,-175.795,7.698,148.255
C07968=1224.060,380.132,-77.078,-175.797,7.695,148.255
C07969=1224.064,379.885,-77.045,-175.798,7.692,148.254
C07970=1224.068,379.637,-77.011,-175.799,7.690,148.254
C07971=1224.072,379.389,-76.978,-175.800,7.688,148.254
C07972=1224.077,379.142,-76.944,-175.801,7.685,148.253
C07973=1224.081,378.894,-76.911,-175.802,7.682,148.253
C07974=1224.085,378.646,-76.877,-175.803,7.679,148.252
C07975=1224.089,378.398,-76.844,-175.804,7.676,148.252
C07976=1224.092,378.151,-76.810,-175.805,7.673,148.252
C07977=1224.097,377.903,-76.777,-175.807,7.671,148.251
C07978=1224.101,377.655,-76.743,-175.807,7.669,148.251
C07979=1224.106,377.407,-76.710,-175.808,7.666,148.250
C07980=1224.110,377.160,-76.677,-175.810,7.663,148.250
C07981=1224.114,376.912,-76.643,-175.811,7.660,148.250
C07982=1224.117,376.664,-76.609,-175.812,7.657,148.249
C07983=1224.121,376.416,-76.576,-175.813,7.655,148.249
C07984=1224.125,376.169,-76.543,-175.815,7.652,148.249
C07985=1224.130,375.921,-76.510,-175.816,7.649,148.248
C07986=1224.134,375.673,-76.475,-175.817,7.646,148.248
C07987=1224.138,375.426,-76.442,-175.818,7.644,148.247
C07988=1224.142,375.178,-76.409,-175.819,7.641,148.247
C07989=1224.147,374.930,-76.376,-175.820,7.639,148.247
C07990=1224.151,374.682,-76.343,-175.821,7.636,148.246
C07991=1224.155,374.435,-76.310,-175.823,7.633,148.246
C07992=1224.159,374.187,-76.277,-175.824,7.631,148.246
C07993=1224.163,373.939,-76.243,-175.825,7.628,148.245
C07994=1224.167,373.691,-76.210,-175.826,7.625,148.245
C07995=1224.170,373.444,-76.176,-175.828,7.622,148.245
C07996=1224.175,373.196,-76.143,-175.829,7.620,148.244
C07997=1224.179,372.948,-76.110,-175.830,7.617,148.244
C07998=1224.183,372.701,-76.077,-175.832,7.614,148.244
C07999=1224.187,372.453,-76.043,-175.833,7.611,148.243
C08000=1224.191,372.205,-76.010,-175.834,7.608,148.243
C08001=1224.195,371.957,-75.977,-175.836,7.606,148.243
C08002=1224.200,371.709,-75.943,-175.837,7.603,148.242
C08003=1224.204,371.462,-75.910,-175.838,7.600,148.242
C08004=1224.208,371.214,-75.877,-175.839,7.597,148.241
C08005=1224.213,370.966,-75.844,-175.841,7.595,148.241
C08006=1224.217,370.718,-75.811,-175.842,7.592,148.241
C08007=1224.221,370.471,-75.778,-175.843,7.589,148.240
C08008=1224.224,370.223,-75.745,-175.845,7.587,148.240
C08009=1224.228,369.976,-75.712,-175.846,7.584,148.240
C08010=1224.233,369.728,-75.679,-175.847,7.581,148.239
C08011=1224.237,369.480,-75.645,-175.849,7.578,148.239
C08012=1224.241,369.232,-75.613,-175.850,7.576,148.239
C08013=1224.245,368.984,-75.580,-175.851,7.573,148.238
C08014=1224.249,368.736,-75.547,-175.853,7.569,148.238
C08015=1224.254,368.489,-75.514,-175.854,7.567,148.238
C08016=1224.258,368.241,-75.480,-175.856,7.564,148.237
C08017=1224.262,367.993,-75.447,-175.857,7.561,148.237
C08018=1224.266,367.745,-75.414,-175.858,7.558,148.237
C08019=1224.271,367.465,-75.377,-175.860,7.556,148.236
C08020=1224.275,367.186,-75.340,-175.862,7.552,148.236
C08021=1224.280,366.906,-75.302,-175.863,7.549,148.236
C08022=1224.285,366.626,-75.265,-175.865,7.546,148.235
C08023=1224.289,366.378,-75.232,-175.866,7.543,148.235
C08024=1224.292,366.131,-75.200,-175.867,7.540,148.235
C08025=1224.297,365.883,-75.167,-175.869,7.538,148.235
C08026=1224.301,365.635,-75.133,-175.870,7.535,148.234
C08027=1224.305,365.387,-75.101,-175.872,7.533,148.234
C08028=1224.309,365.139,-75.068,-175.874,7.529,148.234
C08029=1224.313,364.891,-75.035,-175.875,7.526,148.233
C08030=1224.318,364.644,-75.001,-175.876,7.524,148.233
C08031=1224.321,364.396,-74.970,-175.878,7.521,148.233
C08032=1224.325,364.148,-74.936,-175.879,7.518,148.232
C08033=1224.330,363.901,-74.904,-175.881,7.516,148.232
C08034=1224.334,363.653,-74.871,-175.882,7.513,148.232
C08035=1224.339,363.405,-74.838,-175.884,7.510,148.232
C08036=1224.342,363.157,-74.806,-175.885,7.507,148.231
C08037=1224.346,362.910,-74.772,-175.887,7.504,148.231
C08038=1224.351,362.661,-74.740,-175.888,7.501,148.231
C08039=1224.355,362.414,-74.707,-175.890,7.499,148.230
C08040=1224.359,362.166,-74.674,-175.891,7.496,148.230
C08041=1224.363,361.918,-74.642,-175.893,7.493,148.230
C08042=1224.367,361.670,-74.609,-175.895,7.490,148.230
C08043=1224.371,361.422,-74.575,-175.896,7.487,148.229
C08044=1224.375,361.174,-74.543,-175.898,7.485,148.229
C08045=1224.379,360.927,-74.511,-175.899,7.482,148.229
C08046=1224.384,360.679,-74.478,-175.900,7.479,148.228
C08047=1224.388,360.431,-74.445,-175.903,7.476,148.228
C08048=1224.392,360.183,-74.412,-175.904,7.473,148.228
C08049=1224.396,359.935,-74.380,-175.905,7.471,148.228
C08050=1224.400,359.688,-74.347,-175.907,7.468,148.227
C08051=1224.404,359.439,-74.315,-175.909,7.466,148.227
C08052=1224.408,359.192,-74.282,-175.910,7.462,148.227
C08053=1224.413,358.944,-74.250,-175.912,7.459,148.227
C08054=1224.417,358.697,-74.217,-175.914,7.457,148.226
C08055=1224.422,358.448,-74.184,-175.915,7.454,148.226
C08056=1224.425,358.201,-74.152,-175.916,7.452,148.226
C08057=1224.429,357.952,-74.119,-175.919,7.448,148.226
C08058=1224.433,357.705,-74.086,-175.920,7.446,148.225
C08059=1224.438,357.457,-74.055,-175.921,7.443,148.225
C08060=1224.442,357.210,-74.022,-175.923,7.440,148.225
C08061=1224.446,356.961,-73.989,-175.925,7.437,148.225
C08062=1224.450,356.714,-73.957,-175.927,7.434,148.224
C08063=1224.454,356.465,-73.924,-175.928,7.432,148.224
C08064=1224.458,356.217,-73.892,-175.930,7.429,148.224
C08065=1224.463,355.970,-73.860,-175.931,7.427,148.224
C08066=1224.467,355.722,-73.827,-175.933,7.423,148.223
C08067=1224.471,355.475,-73.795,-175.935,7.421,148.223
C08068=1224.475,355.226,-73.762,-175.936,7.418,148.223
C08069=1224.479,354.978,-73.730,-175.938,7.415,148.223
C08070=1224.483,354.731,-73.697,-175.940,7.412,148.222
C08071=1224.488,354.483,-73.665,-175.942,7.409,148.222
C08072=1224.492,354.235,-73.633,-175.943,7.407,148.222
C08073=1224.496,353.987,-73.600,-175.945,7.404,148.222
C08074=1224.499,353.739,-73.568,-175.947,7.401,148.221
C08075=1224.504,353.491,-73.536,-175.948,7.398,148.221
C08076=1224.509,353.244,-73.503,-175.950,7.396,148.221
C08077=1224.512,352.996,-73.471,-175.952,7.393,148.221
C08078=1224.517,352.747,-73.439,-175.954,7.390,148.221
C08079=1224.521,352.500,-73.407,-175.955,7.387,148.220
C08080=1224.525,352.252,-73.374,-175.957,7.385,148.220
C08081=1224.529,352.004,-73.342,-175.959,7.381,148.220
C08082=1224.533,351.756,-73.310,-175.961,7.379,148.220
C08083=1224.538,351.509,-73.278,-175.962,7.376,148.219
C08084=1224.542,351.260,-73.246,-175.964,7.373,148.219
C08085=1224.545,351.013,-73.213,-175.966,7.370,148.219
C08086=1224.550,350.764,-73.181,-175.967,7.368,148.219
C08087=1224.554,350.517,-73.149,-175.969,7.365,148.219
C08088=1224.559,350.269,-73.117,-175.971,7.363,148.218
C08089=1224.562,350.021,-73.085,-175.973,7.359,148.218
C08090=1224.567,349.773,-73.053,-175.975,7.357,148.218
C08091=1224.571,349.526,-73.020,-175.976,7.354,148.218
C08092=1224.575,349.277,-72.988,-175.978,7.351,148.218
C08093=1224.579,349.029,-72.956,-175.980,7.348,148.217
C08094=1224.584,348.782,-72.924,-175.982,7.346,148.217
C08095=1224.588,348.534,-72.892,-175.983,7.343,148.217
C08096=1224.591,348.285,-72.860,-175.985,7.340,148.217
C08097=1224.596,348.038,-72.828,-175.987,7.337,148.217
C08098=1224.600,347.790,-72.796,-175.989,7.335,148.217
C08099=1224.605,347.541,-72.764,-175.991,7.331,148.216
C08100=1224.609,347.294,-72.733,-175.992,7.329,148.216
C08101=1224.613,347.046,-72.701,-175.994,7.326,148.216
C08102=1224.617,346.798,-72.668,-175.997,7.323,148.216
C08103=1224.621,346.550,-72.637,-175.998,7.321,148.216
C08104=1224.626,346.302,-72.604,-176.000,7.318,148.216
C08105=1224.630,346.054,-72.572,-176.002,7.316,148.215
C08106=1224.634,345.807,-72.541,-176.004,7.312,148.215
C08107=1224.638,345.558,-72.509,-176.005,7.310,148.215
C08108=1224.642,345.310,-72.477,-176.007,7.307,148.215
C08109=1224.646,345.063,-72.445,-176.009,7.304,148.215
C08110=1224.651,344.815,-72.413,-176.011,7.301,148.214
C08111=1224.655,344.567,-72.381,-176.013,7.299,148.214
C08112=1224.659,344.319,-72.349,-176.015,7.296,148.214
C08113=1224.663,344.071,-72.317,-176.017,7.293,148.214
C08114=1224.668,343.824,-72.286,-176.018,7.291,148.214
C08115=1224.672,343.575,-72.254,-176.021,7.287,148.214
C08116=1224.677,343.327,-72.222,-176.022,7.285,148.213
C08117=1224.680,343.079,-72.191,-176.024,7.282,148.213
C08118=1224.684,342.831,-72.159,-176.027,7.279,148.213
C08119=1224.688,342.584,-72.127,-176.028,7.277,148.213
C08120=1224.693,342.335,-72.095,-176.030,7.274,148.213
C08121=1224.697,342.087,-72.064,-176.032,7.271,148.213
C08122=1224.701,341.839,-72.032,-176.034,7.268,148.212
C08123=1224.705,341.562,-71.997,-176.036,7.265,148.212
C08124=1224.710,341.284,-71.960,-176.038,7.263,148.212
C08125=1224.715,341.006,-71.925,-176.040,7.259,148.212
C08126=1224.720,340.729,-71.890,-176.043,7.256,148.212
C08127=1224.724,340.481,-71.858,-176.044,7.254,148.212
C08128=1224.728,340.232,-71.827,-176.046,7.251,148.212
C08129=1224.733,339.985,-71.795,-176.048,7.248,148.211
C08130=1224.736,339.737,-71.763,-176.050,7.246,148.211
C08131=1224.741,339.489,-71.732,-176.052,7.243,148.211
C08132=1224.745,339.241,-71.701,-176.054,7.240,148.211
C08133=1224.750,338.993,-71.669,-176.056,7.237,148.211
C08134=1224.754,338.745,-71.637,-176.058,7.235,148.211
C08135=1224.758,338.497,-71.606,-176.060,7.232,148.211
C08136=1224.762,338.249,-71.574,-176.062,7.229,148.210
C08137=1224.766,338.001,-71.543,-176.064,7.227,148.211
C08138=1224.770,337.753,-71.512,-176.066,7.224,148.210
C08139=1224.774,337.506,-71.480,-176.068,7.221,148.210
C08140=1224.778,337.257,-71.449,-176.070,7.219,148.210
C08141=1224.784,337.009,-71.417,-176.072,7.215,148.210
C08142=1224.788,336.761,-71.386,-176.073,7.213,148.210
C08143=1224.792,336.513,-71.354,-176.076,7.211,148.210
C08144=1224.796,336.265,-71.322,-176.078,7.207,148.210
C08145=1224.800,336.017,-71.292,-176.079,7.205,148.209
C08146=1224.804,335.769,-71.260,-176.082,7.202,148.209
C08147=1224.808,335.521,-71.229,-176.084,7.199,148.209
C08148=1224.812,335.273,-71.197,-176.086,7.197,148.209
C08149=1224.817,335.025,-71.166,-176.088,7.194,148.209
C08150=1224.821,334.777,-71.135,-176.090,7.191,148.209
C08151=1224.825,334.529,-71.104,-176.092,7.189,148.209
C08152=1224.829,334.281,-71.072,-176.094,7.186,148.209
C08153=1224.833,334.033,-71.041,-176.096,7.183,148.209
C08154=1224.837,333.785,-71.009,-176.098,7.181,148.208
C08155=1224.842,333.537,-70.979,-176.100,7.177,148.208
C08156=1224.846,333.289,-70.947,-176.102,7.175,148.208
C08157=1224.850,333.041,-70.916,-176.103,7.173,148.208
C08158=1224.855,332.793,-70.885,-176.106,7.170,148.208
C08159=1224.858,332.545,-70.853,-176.108,7.167,148.208
C08160=1224.863,332.297,-70.823,-176.110,7.165,148.208
C08161=1224.867,332.049,-70.791,-176.112,7.161,148.208
C08162=1224.871,331.801,-70.760,-176.114,7.159,148.208
C08163=1224.875,331.553,-70.729,-176.116,7.156,148.208
C08164=1224.880,331.305,-70.698,-176.118,7.154,148.208
C08165=1224.884,331.058,-70.667,-176.120,7.151,148.207
C08166=1224.888,330.809,-70.636,-176.123,7.148,148.207
C08167=1224.893,330.561,-70.605,-176.124,7.146,148.207
C08168=1224.897,330.313,-70.573,-176.126,7.143,148.207
C08169=1224.901,330.065,-70.542,-176.129,7.140,148.207
C08170=1224.906,329.817,-70.511,-176.131,7.138,148.207
C08171=1224.910,329.568,-70.480,-176.132,7.135,148.207
C08172=1224.913,329.321,-70.449,-176.135,7.132,148.207
C08173=1224.918,329.073,-70.419,-176.137,7.130,148.207
C08174=1224.922,328.825,-70.387,-176.139,7.127,148.207
C08175=1224.927,328.577,-70.357,-176.141,7.124,148.207
C08176=1224.930,328.329,-70.325,-176.143,7.122,148.207
C08177=1224.935,328.081,-70.294,-176.146,7.119,148.207
C08178=1224.940,327.833,-70.263,-176.147,7.116,148.206
C08179=1224.943,327.584,-70.233,-176.149,7.114,148.206
C08180=1224.947,327.336,-70.202,-176.152,7.111,148.206
C08181=1224.952,327.088,-70.171,-176.154,7.108,148.206
C08182=1224.956,326.840,-70.139,-176.156,7.106,148.206
C08183=1224.960,326.592,-70.109,-176.158,7.103,148.206
C08184=1224.965,326.345,-70.078,-176.160,7.101,148.206
C08185=1224.968,326.096,-70.047,-176.162,7.098,148.206
C08186=1224.973,325.848,-70.017,-176.164,7.095,148.206
C08187=1224.978,325.600,-69.986,-176.166,7.093,148.206
C08188=1224.982,325.352,-69.955,-176.169,7.089,148.206
C08189=1224.985,325.104,-69.925,-176.171,7.087,148.206
C08190=1224.990,324.856,-69.894,-176.173,7.085,148.206
C08191=1224.995,324.608,-69.863,-176.175,7.082,148.206
C08192=1224.999,324.359,-69.832,-176.177,7.079,148.206
C08193=1225.003,324.112,-69.802,-176.179,7.077,148.206
C08194=1225.007,323.864,-69.771,-176.181,7.074,148.206
C08195=1225.011,323.615,-69.740,-176.184,7.072,148.206
C08196=1225.016,323.367,-69.709,-176.186,7.069,148.206
C08197=1225.020,323.119,-69.679,-176.188,7.066,148.205
C08198=1225.024,322.872,-69.648,-176.190,7.064,148.205
C08199=1225.028,322.623,-69.617,-176.192,7.062,148.205
C08200=1225.032,322.375,-69.587,-176.194,7.058,148.205
C08201=1225.037,322.127,-69.556,-176.196,7.056,148.205
C08202=1225.041,321.879,-69.525,-176.199,7.053,148.205
C08203=1225.045,321.631,-69.495,-176.201,7.050,148.205
C08204=1225.049,321.383,-69.464,-176.203,7.048,148.205
C08205=1225.054,321.135,-69.433,-176.205,7.045,148.205
C08206=1225.058,320.887,-69.404,-176.207,7.043,148.205
C08207=1225.062,320.638,-69.373,-176.209,7.040,148.205
C08208=1225.067,320.390,-69.342,-176.212,7.037,148.205
C08209=1225.071,320.143,-69.312,-176.214,7.035,148.205
C08210=1225.075,319.895,-69.281,-176.216,7.033,148.205
C08211=1225.078,319.646,-69.250,-176.218,7.030,148.205
C08212=1225.083,319.398,-69.220,-176.220,7.027,148.205
C08213=1225.088,319.150,-69.190,-176.223,7.024,148.205
C08214=1225.092,318.902,-69.159,-176.225,7.022,148.205
C08215=1225.096,318.654,-69.129,-176.227,7.020,148.205
C08216=1225.100,318.405,-69.099,-176.229,7.016,148.205
C08217=1225.105,318.157,-69.068,-176.231,7.014,148.205
C08218=1225.109,317.909,-69.038,-176.234,7.012,148.205
C08219=1225.113,317.662,-69.007,-176.236,7.009,148.205
C08220=1225.117,317.413,-68.978,-176.238,7.007,148.205
C08221=1225.122,317.165,-68.947,-176.240,7.004,148.205
C08222=1225.126,316.917,-68.916,-176.243,7.001,148.205
C08223=1225.130,316.668,-68.886,-176.245,6.999,148.205
C08224=1225.135,316.420,-68.856,-176.247,6.997,148.205
C08225=1225.139,316.173,-68.825,-176.249,6.994,148.205
C08226=1225.144,315.924,-68.795,-176.252,6.991,148.205
C08227=1225.148,315.649,-68.762,-176.254,6.988,148.205
C08228=1225.153,315.372,-68.728,-176.256,6.985,148.205
C08229=1225.157,315.098,-68.695,-176.258,6.983,148.205
C08230=1225.162,314.821,-68.661,-176.261,6.980,148.205
C08231=1225.166,314.573,-68.631,-176.263,6.978,148.205
C08232=1225.171,314.325,-68.601,-176.266,6.974,148.205
C08233=1225.174,314.077,-68.570,-176.268,6.972,148.205
C08234=1225.179,313.829,-68.540,-176.271,6.969,148.205
C08235=1225.183,313.580,-68.510,-176.273,6.967,148.205
C08236=1225.187,313.333,-68.480,-176.275,6.965,148.205
C08237=1225.192,313.084,-68.450,-176.277,6.961,148.205
C08238=1225.196,312.836,-68.420,-176.279,6.959,148.205
C08239=1225.201,312.588,-68.390,-176.281,6.957,148.205
C08240=1225.205,312.340,-68.360,-176.284,6.954,148.205
C08241=1225.209,312.092,-68.330,-176.286,6.952,148.205
C08242=1225.214,311.843,-68.300,-176.288,6.949,148.205
C08243=1225.218,311.596,-68.270,-176.291,6.946,148.205
C08244=1225.222,311.346,-68.240,-176.293,6.944,148.205
C08245=1225.226,311.099,-68.209,-176.295,6.942,148.205
C08246=1225.230,310.851,-68.180,-176.298,6.939,148.205
C08247=1225.235,310.603,-68.149,-176.300,6.937,148.205
C08248=1225.239,310.354,-68.120,-176.302,6.934,148.205
C08249=1225.243,310.106,-68.090,-176.305,6.931,148.205
C08250=1225.248,309.858,-68.060,-176.307,6.929,148.205
C08251=1225.252,309.610,-68.030,-176.309,6.927,148.205
C08252=1225.256,309.362,-68.001,-176.311,6.924,148.205
C08253=1225.261,309.114,-67.970,-176.314,6.922,148.205
C08254=1225.265,308.865,-67.940,-176.316,6.920,148.205
C08255=1225.269,308.617,-67.911,-176.318,6.916,148.205
C08256=1225.273,308.369,-67.881,-176.320,6.914,148.205
C08257=1225.278,308.121,-67.851,-176.322,6.912,148.205
C08258=1225.282,307.873,-67.821,-176.325,6.909,148.205
C08259=1225.286,307.624,-67.792,-176.327,6.906,148.205
C08260=1225.290,307.377,-67.762,-176.329,6.903,148.205
C08261=1225.295,307.128,-67.732,-176.332,6.901,148.205
C08262=1225.299,306.880,-67.702,-176.334,6.899,148.206
C08263=1225.303,306.632,-67.673,-176.337,6.896,148.206
C08264=1225.307,306.383,-67.643,-176.339,6.894,148.206
C08265=1225.312,306.135,-67.612,-176.341,6.892,148.206
C08266=1225.316,305.887,-67.583,-176.344,6.889,148.206
C08267=1225.320,305.639,-67.554,-176.346,6.887,148.206
C08268=1225.325,305.391,-67.524,-176.348,6.884,148.206
C08269=1225.329,305.143,-67.495,-176.351,6.881,148.206
C08270=1225.334,304.895,-67.466,-176.353,6.879,148.206
C08271=1225.339,304.646,-67.436,-176.355,6.877,148.206
C08272=1225.342,304.398,-67.405,-176.357,6.875,148.206
C08273=1225.347,304.150,-67.376,-176.360,6.872,148.206
C08274=1225.351,303.902,-67.346,-176.362,6.869,148.206
C08275=1225.355,303.654,-67.317,-176.364,6.867,148.206
C08276=1225.359,303.405,-67.288,-176.366,6.864,148.206
C08277=1225.363,303.157,-67.258,-176.369,6.862,148.206
C08278=1225.368,302.909,-67.228,-176.371,6.860,148.206
C08279=1225.372,302.660,-67.199,-176.373,6.857,148.206
C08280=1225.377,302.412,-67.169,-176.376,6.855,148.207
C08281=1225.381,302.164,-67.140,-176.378,6.852,148.207
C08282=1225.386,301.916,-67.111,-176.381,6.849,148.207
C08283=1225.390,301.668,-67.081,-176.383,6.847,148.207
C08284=1225.394,301.420,-67.052,-176.385,6.845,148.207
C08285=1225.398,301.171,-67.022,-176.388,6.842,148.207
C08286=1225.402,300.923,-66.993,-176.390,6.840,148.207
C08287=1225.406,300.675,-66.963,-176.392,6.837,148.207
C08288=1225.411,300.427,-66.934,-176.395,6.835,148.207
C08289=1225.415,300.178,-66.904,-176.397,6.833,148.207
C08290=1225.420,299.930,-66.876,-176.399,6.830,148.207
C08291=1225.424,299.682,-66.847,-176.402,6.827,148.207
C08292=1225.428,299.434,-66.817,-176.404,6.825,148.207
C08293=1225.432,299.185,-66.788,-176.406,6.823,148.207
C08294=1225.437,298.937,-66.758,-176.408,6.821,148.207
C08295=1225.441,298.689,-66.729,-176.411,6.818,148.208
C08296=1225.446,298.441,-66.700,-176.413,6.816,148.208
C08297=1225.450,298.192,-66.671,-176.415,6.813,148.208
C08298=1225.454,297.944,-66.642,-176.418,6.810,148.208
C08299=1225.458,297.696,-66.612,-176.420,6.808,148.208
C08300=1225.463,297.448,-66.583,-176.422,6.806,148.208
C08301=1225.467,297.199,-66.553,-176.425,6.803,148.208
C08302=1225.472,296.951,-66.525,-176.428,6.801,148.208
C08303=1225.476,296.703,-66.495,-176.430,6.799,148.208
C08304=1225.480,296.455,-66.466,-176.432,6.796,148.208
C08305=1225.484,296.206,-66.436,-176.434,6.793,148.208
C08306=1225.489,295.957,-66.408,-176.437,6.792,148.209
C08307=1225.493,295.710,-66.379,-176.439,6.789,148.209
C08308=1225.497,295.462,-66.350,-176.442,6.786,148.209
C08309=1225.502,295.213,-66.321,-176.444,6.784,148.209
C08310=1225.506,294.965,-66.292,-176.446,6.782,148.209
C08311=1225.511,294.717,-66.262,-176.449,6.779,148.209
C08312=1225.515,294.468,-66.234,-176.451,6.777,148.209
C08313=1225.519,294.220,-66.204,-176.453,6.775,148.209
C08314=1225.523,293.972,-66.175,-176.456,6.773,148.209
C08315=1225.528,293.724,-66.147,-176.459,6.770,148.209
C08316=1225.532,293.476,-66.118,-176.461,6.768,148.209
C08317=1225.536,293.227,-66.089,-176.463,6.765,148.210
C08318=1225.541,292.978,-66.059,-176.466,6.762,148.210
C08319=1225.545,292.731,-66.030,-176.468,6.760,148.210
C08320=1225.549,292.482,-66.002,-176.470,6.758,148.210
C08321=1225.553,292.234,-65.973,-176.472,6.756,148.210
C08322=1225.558,291.985,-65.944,-176.475,6.753,148.210
C08323=1225.563,291.738,-65.915,-176.478,6.751,148.210
C08324=1225.566,291.489,-65.887,-176.480,6.749,148.210
C08325=1225.571,291.241,-65.857,-176.482,6.746,148.210
C08326=1225.576,290.993,-65.829,-176.485,6.744,148.210
C08327=1225.580,290.744,-65.799,-176.487,6.742,148.211
C08328=1225.584,290.496,-65.771,-176.489,6.739,148.211
C08329=1225.588,290.248,-65.742,-176.492,6.736,148.211
C08330=1225.593,289.999,-65.713,-176.494,6.734,148.211
C08331=1225.598,289.725,-65.682,-176.497,6.732,148.211
C08332=1225.602,289.451,-65.650,-176.499,6.729,148.211
C08333=1225.607,289.177,-65.618,-176.502,6.726,148.211
C08334=1225.612,288.903,-65.587,-176.504,6.724,148.211
C08335=1225.616,288.655,-65.558,-176.508,6.722,148.212
C08336=1225.620,288.406,-65.529,-176.510,6.719,148.212
C08337=1225.625,288.158,-65.501,-176.512,6.717,148.212
C08338=1225.629,287.910,-65.472,-176.514,6.715,148.212
C08339=1225.633,287.661,-65.443,-176.517,6.712,148.212
C08340=1225.638,287.413,-65.415,-176.519,6.710,148.212
C08341=1225.642,287.164,-65.387,-176.522,6.708,148.212
C08342=1225.646,286.916,-65.357,-176.524,6.706,148.212
C08343=1225.651,286.668,-65.329,-176.527,6.703,148.212
C08344=1225.655,286.419,-65.301,-176.529,6.701,148.213
C08345=1225.660,286.171,-65.272,-176.531,6.699,148.213
C08346=1225.664,285.923,-65.243,-176.533,6.696,148.213
C08347=1225.668,285.674,-65.215,-176.537,6.694,148.213
C08348=1225.673,285.426,-65.186,-176.539,6.692,148.213
C08349=1225.677,285.178,-65.158,-176.541,6.689,148.213
C08350=1225.682,284.929,-65.130,-176.543,6.687,148.214
C08351=1225.686,284.682,-65.101,-176.546,6.684,148.214
C08352=1225.691,284.433,-65.072,-176.548,6.682,148.214
C08353=1225.694,284.185,-65.044,-176.551,6.680,148.214
C08354=1225.699,283.936,-65.016,-176.553,6.678,148.214
C08355=1225.703,283.688,-64.988,-176.556,6.675,148.214
C08356=1225.708,283.439,-64.959,-176.558,6.673,148.214
C08357=1225.713,283.192,-64.930,-176.560,6.671,148.214
C08358=1225.716,282.943,-64.902,-176.563,6.669,148.215
C08359=1225.721,282.695,-64.873,-176.565,6.667,148.215
C08360=1225.725,282.446,-64.845,-176.568,6.664,148.215
C08361=1225.730,282.198,-64.817,-176.570,6.662,148.215
C08362=1225.734,281.949,-64.789,-176.572,6.660,148.215
C08363=1225.738,281.701,-64.761,-176.575,6.658,148.215
C08364=1225.743,281.453,-64.732,-176.578,6.655,148.215
C08365=1225.747,281.204,-64.704,-176.580,6.653,148.216
C08366=1225.752,280.956,-64.676,-176.582,6.651,148.216
C08367=1225.755,280.707,-64.648,-176.584,6.648,148.216
C08368=1225.760,280.459,-64.619,-176.587,6.646,148.216
C08369=1225.764,280.211,-64.591,-176.590,6.643,148.216
C08370=1225.769,279.962,-64.563,-176.592,6.642,148.216
C08371=1225.773,279.714,-64.535,-176.594,6.639,148.217
C08372=1225.777,279.466,-64.507,-176.597,6.637,148.217
C08373=1225.782,279.217,-64.478,-176.600,6.634,148.217
C08374=1225.786,278.969,-64.450,-176.602,6.632,148.217
C08375=1225.790,278.721,-64.422,-176.604,6.630,148.217
C08376=1225.795,278.472,-64.394,-176.607,6.628,148.217
C08377=1225.799,278.225,-64.366,-176.609,6.626,148.218
C08378=1225.804,277.976,-64.337,-176.612,6.623,148.218
C08379=1225.809,277.727,-64.310,-176.614,6.621,148.218
C08380=1225.812,277.479,-64.282,-176.617,6.619,148.218
C08381=1225.817,277.230,-64.254,-176.619,6.617,148.218
C08382=1225.821,276.982,-64.226,-176.621,6.615,148.218
C08383=1225.826,276.734,-64.198,-176.624,6.612,148.219
C08384=1225.830,276.485,-64.169,-176.626,6.610,148.219
C08385=1225.835,276.237,-64.142,-176.629,6.608,148.219
C08386=1225.839,275.989,-64.114,-176.631,6.606,148.219
C08387=1225.843,275.740,-64.086,-176.634,6.604,148.219
C08388=1225.848,275.492,-64.058,-176.636,6.601,148.219
C08389=1225.852,275.243,-64.030,-176.639,6.599,148.219
C08390=1225.856,274.995,-64.002,-176.641,6.597,148.220
C08391=1225.861,274.746,-63.974,-176.643,6.595,148.220
C08392=1225.865,274.498,-63.946,-176.646,6.593,148.220
C08393=1225.869,274.250,-63.918,-176.648,6.591,148.220
C08394=1225.874,274.001,-63.891,-176.651,6.588,148.220
C08395=1225.879,273.753,-63.862,-176.653,6.586,148.220
C08396=1225.883,273.505,-63.835,-176.656,6.584,148.221
C08397=1225.887,273.256,-63.807,-176.658,6.581,148.221
C08398=1225.891,273.008,-63.779,-176.661,6.580,148.221
C08399=1225.895,272.759,-63.751,-176.663,6.577,148.221
C08400=1225.901,272.510,-63.724,-176.666,6.575,148.221
C08401=1225.905,272.263,-63.696,-176.668,6.573,148.222
C08402=1225.909,272.013,-63.668,-176.671,6.571,148.222
C08403=1225.913,271.766,-63.641,-176.673,6.569,148.222
C08404=1225.918,271.518,-63.613,-176.675,6.566,148.222
C08405=1225.922,271.268,-63.585,-176.678,6.564,148.222
C08406=1225.927,271.020,-63.557,-176.681,6.562,148.222
C08407=1225.931,270.772,-63.530,-176.683,6.560,148.223
C08408=1225.935,270.523,-63.502,-176.685,6.557,148.223
C08409=1225.940,270.275,-63.475,-176.688,6.556,148.223
C08410=1225.944,270.027,-63.447,-176.690,6.553,148.223
C08411=1225.948,269.778,-63.420,-176.693,6.551,148.223
C08412=1225.953,269.530,-63.392,-176.695,6.548,148.224
C08413=1225.957,269.281,-63.365,-176.698,6.546,148.224
C08414=1225.962,269.032,-63.336,-176.701,6.545,148.224
C08415=1225.966,268.784,-63.309,-176.703,6.542,148.224
C08416=1225.971,268.536,-63.281,-176.705,6.541,148.224
C08417=1225.975,268.288,-63.254,-176.707,6.538,148.225
C08418=1225.979,268.039,-63.226,-176.711,6.536,148.225
C08419=1225.984,267.790,-63.199,-176.713,6.533,148.225
C08420=1225.988,267.543,-63.171,-176.715,6.531,148.225
C08421=1225.993,267.294,-63.144,-176.718,6.530,148.225
C08422=1225.997,267.045,-63.117,-176.720,6.527,148.226
C08423=1226.001,266.797,-63.089,-176.723,6.525,148.226
C08424=1226.006,266.549,-63.062,-176.725,6.523,148.226
C08425=1226.011,266.300,-63.035,-176.728,6.521,148.226
C08426=1226.014,266.051,-63.007,-176.730,6.518,148.226
C08427=1226.019,265.803,-62.980,-176.733,6.516,148.227
C08428=1226.024,265.554,-62.952,-176.735,6.515,148.227
C08429=1226.028,265.307,-62.925,-176.737,6.512,148.227
C08430=1226.032,265.057,-62.897,-176.740,6.510,148.227
C08431=1226.037,264.809,-62.870,-176.742,6.508,148.227
C08432=1226.041,264.561,-62.842,-176.745,6.506,148.228
C08433=1226.046,264.313,-62.815,-176.748,6.504,148.228
C08434=1226.050,264.064,-62.788,-176.750,6.501,148.228
C08435=1226.054,263.791,-62.758,-176.753,6.500,148.228
C08436=1226.059,263.518,-62.728,-176.756,6.497,148.228
C08437=1226.064,263.246,-62.698,-176.758,6.495,148.229
C08438=1226.070,262.973,-62.669,-176.760,6.493,148.229
C08439=1226.074,262.725,-62.641,-176.763,6.491,148.229
C08440=1226.079,262.476,-62.614,-176.766,6.488,148.229
C08441=1226.083,262.228,-62.587,-176.768,6.486,148.230
C08442=1226.087,261.979,-62.560,-176.771,6.484,148.230
C08443=1226.091,261.731,-62.533,-176.773,6.482,148.230
C08444=1226.096,261.482,-62.506,-176.776,6.480,148.230
C08445=1226.101,261.234,-62.479,-176.778,6.478,148.230
C08446=1226.105,260.986,-62.451,-176.780,6.476,148.231
C08447=1226.110,260.737,-62.424,-176.783,6.474,148.231
C08448=1226.113,260.488,-62.397,-176.786,6.472,148.231
C08449=1226.118,260.240,-62.370,-176.788,6.469,148.231
C08450=1226.122,259.991,-62.343,-176.791,6.467,148.232
C08451=1226.127,259.743,-62.316,-176.793,6.465,148.232
C08452=1226.131,259.494,-62.289,-176.796,6.463,148.232
C08453=1226.136,259.246,-62.262,-176.798,6.461,148.232
C08454=1226.140,258.998,-62.235,-176.801,6.459,148.233
C08455=1226.145,258.749,-62.208,-176.803,6.457,148.233
C08456=1226.149,258.500,-62.181,-176.806,6.455,148.233
C08457=1226.153,258.251,-62.154,-176.808,6.453,148.233
C08458=1226.157,258.003,-62.127,-176.810,6.451,148.233
C08459=1226.162,257.755,-62.100,-176.813,6.449,148.234
C08460=1226.167,257.506,-62.073,-176.816,6.447,148.234
C08461=1226.171,257.258,-62.046,-176.818,6.444,148.234
C08462=1226.175,257.010,-62.020,-176.821,6.442,148.234
C08463=1226.180,256.761,-61.993,-176.823,6.441,148.235
C08464=1226.185,256.513,-61.965,-176.825,6.438,148.235
C08465=1226.189,256.264,-61.938,-176.828,6.436,148.235
C08466=1226.193,256.015,-61.913,-176.831,6.435,148.235
C08467=1226.198,255.767,-61.886,-176.833,6.432,148.235
C08468=1226.202,255.518,-61.858,-176.835,6.431,148.236
C08469=1226.206,255.269,-61.832,-176.838,6.429,148.236
C08470=1226.211,255.021,-61.805,-176.840,6.426,148.236
C08471=1226.215,254.772,-61.778,-176.843,6.425,148.236
C08472=1226.219,254.524,-61.751,-176.845,6.423,148.237
C08473=1226.224,254.275,-61.725,-176.848,6.421,148.237
C08474=1226.229,254.027,-61.698,-176.851,6.418,148.237
C08475=1226.233,253.778,-61.671,-176.853,6.416,148.237
C08476=1226.237,253.530,-61.644,-176.856,6.414,148.238
C08477=1226.242,253.281,-61.617,-176.858,6.412,148.238
C08478=1226.246,253.033,-61.591,-176.861,6.410,148.238
C08479=1226.251,252.784,-61.564,-176.863,6.408,148.238
C08480=1226.255,252.536,-61.538,-176.866,6.406,148.239
C08481=1226.260,252.288,-61.511,-176.868,6.404,148.239
C08482=1226.265,252.038,-61.484,-176.871,6.402,148.239
C08483=1226.268,251.790,-61.458,-176.873,6.400,148.239
C08484=1226.273,251.542,-61.431,-176.875,6.398,148.239
C08485=1226.277,251.293,-61.405,-176.878,6.396,148.240
C08486=1226.282,251.044,-61.378,-176.881,6.394,148.240
C08487=1226.286,250.796,-61.352,-176.883,6.392,148.240
C08488=1226.291,250.547,-61.325,-176.885,6.390,148.240
C08489=1226.295,250.299,-61.299,-176.888,6.388,148.241
C08490=1226.299,250.050,-61.272,-176.891,6.386,148.241
C08491=1226.304,249.801,-61.245,-176.893,6.384,148.241
C08492=1226.308,249.553,-61.219,-176.895,6.382,148.241
C08493=1226.314,249.305,-61.193,-176.898,6.380,148.242
C08494=1226.318,249.057,-61.166,-176.900,6.379,148.242
C08495=1226.323,248.807,-61.140,-176.903,6.377,148.242
C08496=1226.327,248.559,-61.114,-176.905,6.374,148.242
C08497=1226.331,248.311,-61.087,-176.908,6.373,148.243
C08498=1226.336,248.062,-61.061,-176.910,6.371,148.243
C08499=1226.340,247.814,-61.034,-176.914,6.368,148.243
C08500=1226.344,247.565,-61.008,-176.916,6.366,148.243
C08501=1226.348,247.316,-60.982,-176.918,6.364,148.244
C08502=1226.353,247.067,-60.955,-176.921,6.362,148.244
C08503=1226.357,246.819,-60.929,-176.924,6.360,148.244
C08504=1226.362,246.570,-60.902,-176.926,6.358,148.244
C08505=1226.367,246.323,-60.876,-176.928,6.356,148.245
C08506=1226.372,246.073,-60.850,-176.931,6.354,148.245
C08507=1226.376,245.825,-60.824,-176.934,6.352,148.245
C08508=1226.380,245.576,-60.798,-176.936,6.350,148.245
C08509=1226.385,245.327,-60.771,-176.938,6.348,148.246
C08510=1226.389,245.079,-60.745,-176.941,6.346,148.246
C08511=1226.393,244.830,-60.719,-176.944,6.344,148.246
C08512=1226.398,244.581,-60.693,-176.946,6.343,148.247
C08513=1226.402,244.334,-60.667,-176.948,6.340,148.247
C08514=1226.407,244.085,-60.640,-176.951,6.339,148.247
C08515=1226.411,243.836,-60.614,-176.954,6.337,148.247
C08516=1226.416,243.588,-60.588,-176.956,6.335,148.248
C08517=1226.421,243.339,-60.562,-176.959,6.333,148.248
C08518=1226.424,243.090,-60.535,-176.961,6.331,148.248
C08519=1226.429,242.842,-60.510,-176.963,6.329,148.248
C08520=1226.434,242.593,-60.484,-176.966,6.327,148.249
C08521=1226.438,242.344,-60.458,-176.969,6.325,148.249
C08522=1226.442,242.096,-60.431,-176.971,6.323,148.249
C08523=1226.447,241.847,-60.406,-176.973,6.321,148.249
C08524=1226.452,241.598,-60.379,-176.976,6.319,148.250
C08525=1226.456,241.350,-60.354,-176.979,6.317,148.250
C08526=1226.460,241.102,-60.327,-176.981,6.315,148.250
C08527=1226.465,240.853,-60.301,-176.984,6.313,148.251
C08528=1226.470,240.604,-60.275,-176.986,6.311,148.251
C08529=1226.474,240.356,-60.250,-176.989,6.309,148.251
C08530=1226.479,240.107,-60.224,-176.991,6.308,148.251
C08531=1226.482,239.859,-60.198,-176.993,6.307,148.252
C08532=1226.487,239.610,-60.171,-176.996,6.305,148.252
C08533=1226.492,239.361,-60.146,-176.999,6.303,148.252
C08534=1226.496,239.113,-60.120,-177.001,6.301,148.252
C08535=1226.501,238.864,-60.095,-177.003,6.299,148.253
C08536=1226.506,238.615,-60.068,-177.006,6.297,148.253
C08537=1226.510,238.366,-60.042,-177.009,6.295,148.253
C08538=1226.514,238.119,-60.016,-177.011,6.293,148.254
C08539=1226.519,237.847,-59.988,-177.014,6.290,148.254
C08540=1226.524,237.575,-59.960,-177.017,6.288,148.254
C08541=1226.529,237.304,-59.932,-177.020,6.287,148.255
C08542=1226.533,237.032,-59.904,-177.022,6.285,148.255
C08543=1226.538,236.784,-59.878,-177.025,6.283,148.255
C08544=1226.543,236.535,-59.853,-177.027,6.281,148.256
C08545=1226.548,236.286,-59.826,-177.030,6.279,148.256
C08546=1226.552,236.038,-59.801,-177.032,6.277,148.256
C08547=1226.557,235.789,-59.775,-177.035,6.275,148.256
C08548=1226.561,235.541,-59.749,-177.037,6.273,148.257
C08549=1226.565,235.292,-59.724,-177.040,6.271,148.257
C08550=1226.570,235.044,-59.698,-177.043,6.269,148.257
C08551=1226.574,234.795,-59.673,-177.045,6.268,148.258
C08552=1226.578,234.546,-59.647,-177.047,6.265,148.258
C08553=1226.583,234.298,-59.621,-177.050,6.263,148.258
C08554=1226.587,234.049,-59.596,-177.053,6.262,148.258
C08555=1226.592,233.800,-59.571,-177.055,6.260,148.259
C08556=1226.597,233.551,-59.545,-177.058,6.258,148.259
C08557=1226.602,233.303,-59.519,-177.061,6.256,148.259
C08558=1226.606,233.054,-59.493,-177.063,6.255,148.260
C08559=1226.611,232.806,-59.468,-177.065,6.253,148.260
C08560=1226.615,232.557,-59.442,-177.067,6.251,148.260
C08561=1226.619,232.308,-59.416,-177.070,6.249,148.260
C08562=1226.624,232.060,-59.391,-177.073,6.247,148.261
C08563=1226.629,231.811,-59.366,-177.075,6.245,148.261
C08564=1226.633,231.562,-59.340,-177.078,6.243,148.261
C08565=1226.638,231.314,-59.315,-177.080,6.242,148.262
C08566=1226.642,231.065,-59.289,-177.083,6.240,148.262
C08567=1226.647,230.817,-59.264,-177.086,6.238,148.262
C08568=1226.651,230.567,-59.239,-177.088,6.236,148.263
C08569=1226.655,230.319,-59.213,-177.090,6.234,148.263
C08570=1226.659,230.071,-59.188,-177.093,6.232,148.263
C08571=1226.664,229.822,-59.162,-177.096,6.230,148.263
C08572=1226.669,229.573,-59.138,-177.098,6.228,148.264
C08573=1226.673,229.324,-59.112,-177.100,6.227,148.264
C08574=1226.677,229.076,-59.086,-177.103,6.225,148.264
C08575=1226.682,228.827,-59.061,-177.106,6.223,148.265
C08576=1226.687,228.578,-59.036,-177.108,6.222,148.265
C08577=1226.691,228.330,-59.010,-177.111,6.220,148.265
C08578=1226.696,228.081,-58.985,-177.114,6.218,148.266
C08579=1226.701,227.832,-58.960,-177.116,6.216,148.266
C08580=1226.705,227.584,-58.934,-177.119,6.214,148.266
C08581=1226.709,227.335,-58.910,-177.121,6.212,148.266
C08582=1226.714,227.086,-58.884,-177.124,6.210,148.267
C08583=1226.718,226.837,-58.859,-177.126,6.208,148.267
C08584=1226.723,226.589,-58.834,-177.129,6.206,148.267
C08585=1226.727,226.340,-58.808,-177.131,6.205,148.268
C08586=1226.732,226.091,-58.783,-177.133,6.203,148.268
C08587=1226.736,225.843,-58.758,-177.136,6.201,148.268
C08588=1226.741,225.594,-58.734,-177.139,6.200,148.269
C08589=1226.745,225.345,-58.708,-177.141,6.198,148.269
C08590=1226.750,225.097,-58.683,-177.144,6.196,148.269
C08591=1226.755,224.848,-58.657,-177.147,6.194,148.270
C08592=1226.759,224.599,-58.633,-177.149,6.192,148.270
C08593=1226.763,224.351,-58.608,-177.152,6.190,148.270
C08594=1226.768,224.102,-58.583,-177.154,6.188,148.271
C08595=1226.773,223.853,-58.557,-177.157,6.187,148.271
C08596=1226.778,223.604,-58.533,-177.159,6.186,148.271
C08597=1226.781,223.356,-58.507,-177.162,6.184,148.272
C08598=1226.786,223.107,-58.483,-177.164,6.182,148.272
C08599=1226.791,222.858,-58.457,-177.167,6.180,148.272
C08600=1226.796,222.610,-58.432,-177.169,6.178,148.272
C08601=1226.799,222.361,-58.407,-177.172,6.176,148.273
C08602=1226.804,222.112,-58.382,-177.174,6.174,148.273
C08603=1226.809,221.863,-58.357,-177.177,6.172,148.273
C08604=1226.813,221.615,-58.333,-177.180,6.170,148.274
C08605=1226.818,221.366,-58.308,-177.182,6.169,148.274
C08606=1226.823,221.117,-58.283,-177.184,6.167,148.274
C08607=1226.827,220.869,-58.258,-177.187,6.166,148.275
C08608=1226.831,220.620,-58.233,-177.190,6.164,148.275
C08609=1226.836,220.371,-58.208,-177.192,6.162,148.275
C08610=1226.840,220.123,-58.183,-177.195,6.160,148.276
C08611=1226.845,219.874,-58.159,-177.198,6.158,148.276
C08612=1226.850,219.625,-58.134,-177.200,6.156,148.276
C08613=1226.854,219.377,-58.109,-177.203,6.154,148.277
C08614=1226.859,219.128,-58.084,-177.205,6.153,148.277
C08615=1226.863,218.878,-58.059,-177.207,6.151,148.277
C08616=1226.868,218.630,-58.035,-177.210,6.150,148.278
C08617=1226.872,218.382,-58.010,-177.213,6.148,148.278
C08618=1226.876,218.133,-57.985,-177.215,6.146,148.278
C08619=1226.881,217.884,-57.961,-177.218,6.144,148.279
C08620=1226.886,217.635,-57.935,-177.221,6.142,148.279
C08621=1226.890,217.386,-57.911,-177.223,6.140,148.279
C08622=1226.895,217.138,-57.886,-177.225,6.139,148.280
C08623=1226.899,216.889,-57.862,-177.228,6.137,148.280
C08624=1226.904,216.640,-57.837,-177.231,6.136,148.280
C08625=1226.908,216.392,-57.813,-177.233,6.134,148.281
C08626=1226.913,216.142,-57.788,-177.236,6.132,148.281
C08627=1226.918,215.894,-57.763,-177.238,6.130,148.281
C08628=1226.922,215.645,-57.738,-177.241,6.128,148.282
C08629=1226.927,215.397,-57.713,-177.243,6.127,148.282
C08630=1226.931,215.148,-57.689,-177.246,6.125,148.282
C08631=1226.936,214.899,-57.664,-177.248,6.123,148.283
C08632=1226.940,214.650,-57.640,-177.251,6.121,148.283
C08633=1226.945,214.402,-57.615,-177.254,6.120,148.283
C08634=1226.949,214.152,-57.591,-177.256,6.118,148.284
C08635=1226.954,213.904,-57.566,-177.259,6.116,148.284
C08636=1226.958,213.655,-57.542,-177.261,6.115,148.285
C08637=1226.964,213.407,-57.518,-177.264,6.113,148.285
C08638=1226.967,213.157,-57.493,-177.267,6.111,148.285
C08639=1226.972,212.909,-57.469,-177.269,6.110,148.286
C08640=1226.977,212.660,-57.444,-177.272,6.108,148.286
C08641=1226.981,212.411,-57.420,-177.275,6.106,148.286
C08642=1226.986,212.163,-57.395,-177.277,6.104,148.287
C08643=1226.991,211.892,-57.369,-177.280,6.102,148.287
C08644=1226.995,211.623,-57.342,-177.283,6.100,148.287
C08645=1227.000,211.351,-57.316,-177.285,6.098,148.288
C08646=1227.005,211.081,-57.289,-177.288,6.097,148.288
C08647=1227.010,210.832,-57.265,-177.291,6.095,148.289
C08648=1227.015,210.584,-57.241,-177.294,6.093,148.289
C08649=1227.019,210.335,-57.216,-177.296,6.092,148.289
C08650=1227.024,210.086,-57.192,-177.298,6.090,148.290
C08651=1227.028,209.837,-57.167,-177.301,6.088,148.290
C08652=1227.033,209.588,-57.144,-177.304,6.087,148.290
C08653=1227.038,209.340,-57.119,-177.306,6.085,148.291
C08654=1227.042,209.091,-57.095,-177.309,6.083,148.291
C08655=1227.046,208.842,-57.071,-177.311,6.082,148.291
C08656=1227.051,208.593,-57.046,-177.314,6.080,148.292
C08657=1227.056,208.345,-57.022,-177.316,6.078,148.292
C08658=1227.060,208.095,-56.998,-177.319,6.076,148.292
C08659=1227.065,207.847,-56.974,-177.321,6.074,148.293
C08660=1227.069,207.598,-56.950,-177.323,6.073,148.293
C08661=1227.074,207.350,-56.926,-177.327,6.072,148.294
C08662=1227.079,207.100,-56.902,-177.329,6.070,148.294
C08663=1227.083,206.851,-56.877,-177.332,6.068,148.294
C08664=1227.087,206.603,-56.853,-177.335,6.066,148.295
C08665=1227.092,206.354,-56.829,-177.337,6.065,148.295
C08666=1227.097,206.105,-56.805,-177.339,6.063,148.295
C08667=1227.102,205.857,-56.781,-177.342,6.062,148.296
C08668=1227.106,205.608,-56.757,-177.344,6.060,148.296
C08669=1227.110,205.359,-56.733,-177.347,6.058,148.296
C08670=1227.115,205.110,-56.709,-177.349,6.057,148.297
C08671=1227.120,204.861,-56.685,-177.352,6.055,148.297
C08672=1227.124,204.612,-56.661,-177.354,6.053,148.297
C08673=1227.129,204.364,-56.637,-177.358,6.052,148.298
C08674=1227.133,204.116,-56.613,-177.360,6.050,148.298
C08675=1227.138,203.866,-56.589,-177.362,6.049,148.299
C08676=1227.142,203.617,-56.565,-177.365,6.047,148.299
C08677=1227.147,203.368,-56.541,-177.368,6.045,148.299
C08678=1227.151,203.120,-56.517,-177.370,6.043,148.300
C08679=1227.156,202.871,-56.493,-177.373,6.041,148.300
C08680=1227.161,202.622,-56.470,-177.375,6.040,148.300
C08681=1227.166,202.374,-56.445,-177.378,6.038,148.301
C08682=1227.170,202.124,-56.422,-177.380,6.037,148.301
C08683=1227.175,201.876,-56.398,-177.383,6.035,148.302
C08684=1227.179,201.626,-56.374,-177.385,6.034,148.302
C08685=1227.183,201.378,-56.350,-177.388,6.032,148.302
C08686=1227.188,201.129,-56.327,-177.391,6.030,148.303
C08687=1227.192,200.880,-56.302,-177.393,6.029,148.303
C08688=1227.197,200.631,-56.279,-177.396,6.027,148.303
C08689=1227.202,200.383,-56.254,-177.398,6.026,148.304
C08690=1227.207,200.134,-56.231,-177.401,6.024,148.304
C08691=1227.211,199.885,-56.207,-177.403,6.022,148.304
C08692=1227.216,199.636,-56.184,-177.406,6.020,148.305
C08693=1227.220,199.388,-56.160,-177.409,6.019,148.305
C08694=1227.225,199.139,-56.136,-177.411,6.018,148.306
C08695=1227.230,198.890,-56.113,-177.414,6.016,148.306
C08696=1227.234,198.641,-56.089,-177.416,6.014,148.306
C08697=1227.239,198.392,-56.065,-177.419,6.013,148.307
C08698=1227.243,198.143,-56.041,-177.421,6.011,148.307
C08699=1227.247,197.894,-56.018,-177.424,6.009,148.307
C08700=1227.252,197.645,-55.994,-177.427,6.008,148.308
C08701=1227.256,197.397,-55.970,-177.429,6.007,148.308
C08702=1227.261,197.148,-55.947,-177.432,6.005,148.309
C08703=1227.266,196.899,-55.923,-177.434,6.003,148.309
C08704=1227.270,196.650,-55.899,-177.437,6.001,148.309
C08705=1227.275,196.401,-55.876,-177.439,6.000,148.310
C08706=1227.280,196.152,-55.853,-177.442,5.998,148.310
C08707=1227.284,195.904,-55.829,-177.445,5.997,148.311
C08708=1227.289,195.655,-55.805,-177.447,5.995,148.311
C08709=1227.293,195.406,-55.782,-177.450,5.994,148.311
C08710=1227.298,195.157,-55.758,-177.452,5.992,148.312
C08711=1227.303,194.908,-55.734,-177.455,5.990,148.312
C08712=1227.307,194.659,-55.711,-177.457,5.989,148.312
C08713=1227.312,194.410,-55.688,-177.460,5.987,148.313
C08714=1227.317,194.161,-55.664,-177.463,5.986,148.313
C08715=1227.322,193.913,-55.641,-177.465,5.984,148.314
C08716=1227.326,193.664,-55.617,-177.467,5.983,148.314
C08717=1227.330,193.416,-55.595,-177.470,5.981,148.314
C08718=1227.335,193.167,-55.571,-177.473,5.979,148.315
C08719=1227.340,192.918,-55.548,-177.475,5.977,148.315
C08720=1227.344,192.669,-55.524,-177.478,5.977,148.316
C08721=1227.349,192.420,-55.501,-177.481,5.975,148.316
C08722=1227.354,192.171,-55.477,-177.483,5.973,148.316
C08723=1227.358,191.922,-55.454,-177.485,5.972,148.317
C08724=1227.363,191.673,-55.430,-177.488,5.970,148.317
C08725=1227.367,191.424,-55.408,-177.491,5.968,148.317
C08726=1227.372,191.175,-55.384,-177.493,5.968,148.318
C08727=1227.376,190.926,-55.361,-177.496,5.966,148.318
C08728=1227.381,190.677,-55.337,-177.498,5.964,148.319
C08729=1227.386,190.429,-55.314,-177.501,5.962,148.319
C08730=1227.391,190.180,-55.291,-177.503,5.961,148.320
C08731=1227.395,189.931,-55.268,-177.506,5.959,148.320
C08732=1227.400,189.682,-55.245,-177.509,5.958,148.320
C08733=1227.404,189.433,-55.222,-177.511,5.957,148.321
C08734=1227.409,189.184,-55.198,-177.514,5.955,148.321
C08735=1227.414,188.935,-55.175,-177.516,5.953,148.321
C08736=1227.418,188.686,-55.152,-177.518,5.952,148.322
C08737=1227.422,188.437,-55.129,-177.521,5.950,148.322
C08738=1227.428,188.189,-55.106,-177.524,5.949,148.323
C08739=1227.432,187.940,-55.082,-177.526,5.948,148.323
C08740=1227.436,187.691,-55.060,-177.529,5.946,148.324
C08741=1227.441,187.442,-55.036,-177.532,5.944,148.324
C08742=1227.446,187.193,-55.013,-177.534,5.942,148.324
C08743=1227.450,186.944,-54.990,-177.537,5.941,148.325
C08744=1227.454,186.695,-54.967,-177.539,5.940,148.325
C08745=1227.460,186.447,-54.944,-177.542,5.938,148.326
C08746=1227.465,186.197,-54.921,-177.544,5.937,148.326
C08747=1227.469,185.929,-54.896,-177.547,5.935,148.326
C08748=1227.474,185.659,-54.871,-177.550,5.933,148.327
C08749=1227.480,185.389,-54.846,-177.553,5.931,148.327
C08750=1227.484,185.120,-54.822,-177.556,5.930,148.328
C08751=1227.489,184.871,-54.798,-177.558,5.929,148.328
C08752=1227.494,184.621,-54.776,-177.560,5.927,148.328
C08753=1227.498,184.372,-54.753,-177.563,5.925,148.329
C08754=1227.503,184.123,-54.729,-177.566,5.925,148.329
C08755=1227.508,183.875,-54.706,-177.568,5.923,148.330
C08756=1227.512,183.626,-54.684,-177.571,5.921,148.330
C08757=1227.517,183.376,-54.661,-177.573,5.920,148.331
C08758=1227.521,183.128,-54.638,-177.576,5.918,148.331
C08759=1227.526,182.879,-54.615,-177.579,5.917,148.331
C08760=1227.531,182.630,-54.592,-177.581,5.916,148.332
C08761=1227.535,182.381,-54.570,-177.584,5.914,148.332
C08762=1227.540,182.132,-54.546,-177.586,5.912,148.333
C08763=1227.544,181.883,-54.524,-177.589,5.911,148.333
C08764=1227.549,181.634,-54.501,-177.591,5.909,148.334
C08765=1227.553,181.386,-54.479,-177.594,5.907,148.334
C08766=1227.558,181.137,-54.455,-177.596,5.906,148.334
C08767=1227.563,180.887,-54.433,-177.599,5.905,148.335
C08768=1227.568,180.639,-54.410,-177.601,5.904,148.335
C08769=1227.572,180.390,-54.387,-177.604,5.902,148.336
C08770=1227.577,180.141,-54.365,-177.607,5.900,148.336
C08771=1227.581,179.891,-54.341,-177.609,5.900,148.337
C08772=1227.586,179.643,-54.319,-177.612,5.898,148.337
C08773=1227.591,179.394,-54.296,-177.615,5.896,148.337
C08774=1227.595,179.145,-54.274,-177.617,5.895,148.338
C08775=1227.600,178.896,-54.251,-177.620,5.893,148.338
C08776=1227.604,178.647,-54.229,-177.622,5.892,148.339
C08777=1227.609,178.398,-54.205,-177.625,5.891,148.339
C08778=1227.614,178.150,-54.184,-177.627,5.889,148.339
C08779=1227.619,177.901,-54.160,-177.630,5.888,148.340
C08780=1227.623,177.651,-54.138,-177.632,5.886,148.340
C08781=1227.628,177.402,-54.115,-177.635,5.884,148.341
C08782=1227.632,177.154,-54.093,-177.637,5.883,148.341
C08783=1227.636,176.905,-54.070,-177.640,5.882,148.342
C08784=1227.641,176.655,-54.048,-177.642,5.881,148.342
C08785=1227.646,176.407,-54.025,-177.645,5.879,148.342
C08786=1227.651,176.158,-54.003,-177.648,5.877,148.343
C08787=1227.655,175.909,-53.980,-177.650,5.877,148.343
C08788=1227.661,175.660,-53.958,-177.653,5.875,148.344
C08789=1227.665,175.411,-53.935,-177.655,5.874,148.344
C08790=1227.669,175.163,-53.913,-177.658,5.872,148.344
C08791=1227.674,174.913,-53.891,-177.661,5.870,148.345
C08792=1227.678,174.664,-53.868,-177.663,5.869,148.345
C08793=1227.684,174.415,-53.846,-177.666,5.868,148.346
C08794=1227.688,174.167,-53.823,-177.668,5.867,148.346
C08795=1227.692,173.917,-53.801,-177.671,5.865,148.347
C08796=1227.698,173.668,-53.778,-177.673,5.863,148.347
C08797=1227.702,173.420,-53.756,-177.675,5.862,148.347
C08798=1227.707,173.171,-53.734,-177.679,5.861,148.348
C08799=1227.712,172.921,-53.711,-177.681,5.860,148.348
C08800=1227.716,172.673,-53.689,-177.683,5.858,148.349
C08801=1227.720,172.424,-53.667,-177.687,5.856,148.349
C08802=1227.726,172.174,-53.644,-177.689,5.855,148.350
C08803=1227.730,171.926,-53.622,-177.691,5.854,148.350
C08804=1227.734,171.677,-53.600,-177.693,5.853,148.350
C08805=1227.739,171.427,-53.577,-177.697,5.851,148.351
C08806=1227.744,171.179,-53.555,-177.699,5.849,148.351
C08807=1227.748,170.930,-53.533,-177.701,5.848,148.352
C08808=1227.753,170.681,-53.511,-177.704,5.847,148.352
C08809=1227.758,170.432,-53.488,-177.706,5.846,148.353
C08810=1227.763,170.183,-53.467,-177.709,5.844,148.353
C08811=1227.767,169.934,-53.444,-177.711,5.843,148.354
C08812=1227.772,169.685,-53.422,-177.714,5.841,148.354
C08813=1227.777,169.436,-53.400,-177.716,5.840,148.354
C08814=1227.781,169.187,-53.378,-177.719,5.839,148.355
C08815=1227.786,168.938,-53.356,-177.722,5.837,148.355
C08816=1227.790,168.689,-53.333,-177.724,5.836,148.356
C08817=1227.795,168.440,-53.311,-177.727,5.834,148.356
C08818=1227.800,168.191,-53.289,-177.730,5.834,148.357
C08819=1227.805,167.942,-53.267,-177.732,5.832,148.357
C08820=1227.809,167.693,-53.245,-177.734,5.831,148.358
C08821=1227.814,167.444,-53.223,-177.738,5.829,148.358
C08822=1227.819,167.195,-53.201,-177.740,5.827,148.358
C08823=1227.823,166.947,-53.178,-177.742,5.826,148.359
C08824=1227.828,166.697,-53.156,-177.745,5.825,148.359
C08825=1227.832,166.449,-53.135,-177.748,5.824,148.360
C08826=1227.837,166.199,-53.113,-177.750,5.822,148.360
C08827=1227.842,165.951,-53.091,-177.752,5.821,148.361
C08828=1227.847,165.701,-53.068,-177.755,5.820,148.361
C08829=1227.851,165.452,-53.047,-177.758,5.819,148.362
C08830=1227.856,165.203,-53.025,-177.760,5.817,148.362
C08831=1227.861,164.954,-53.003,-177.763,5.816,148.363
C08832=1227.865,164.705,-52.981,-177.765,5.814,148.363
C08833=1227.870,164.456,-52.959,-177.767,5.813,148.363
C08834=1227.875,164.208,-52.937,-177.771,5.812,148.364
C08835=1227.879,163.958,-52.915,-177.773,5.810,148.364
C08836=1227.884,163.710,-52.894,-177.775,5.809,148.365
C08837=1227.889,163.460,-52.871,-177.779,5.807,148.365
C08838=1227.894,163.212,-52.849,-177.781,5.806,148.366
C08839=1227.898,162.962,-52.827,-177.783,5.805,148.366
C08840=1227.903,162.714,-52.806,-177.786,5.804,148.367
C08841=1227.907,162.464,-52.784,-177.789,5.802,148.367
C08842=1227.912,162.216,-52.762,-177.791,5.801,148.368
C08843=1227.917,161.967,-52.740,-177.794,5.800,148.368
C08844=1227.921,161.717,-52.719,-177.796,5.799,148.368
C08845=1227.926,161.468,-52.697,-177.799,5.797,148.369
C08846=1227.930,161.219,-52.675,-177.801,5.796,148.369
C08847=1227.935,160.970,-52.653,-177.804,5.794,148.370
C08848=1227.940,160.722,-52.632,-177.806,5.794,148.370
C08849=1227.944,160.472,-52.610,-177.809,5.792,148.371
C08850=1227.949,160.224,-52.588,-177.811,5.791,148.371
C08851=1227.955,159.954,-52.565,-177.814,5.789,148.372
C08852=1227.960,159.685,-52.542,-177.817,5.787,148.372
C08853=1227.965,159.417,-52.518,-177.820,5.787,148.373
C08854=1227.969,159.148,-52.495,-177.823,5.785,148.373
C08855=1227.974,158.898,-52.473,-177.825,5.784,148.374
C08856=1227.979,158.650,-52.451,-177.827,5.783,148.374
C08857=1227.983,158.400,-52.430,-177.831,5.781,148.375
C08858=1227.988,158.151,-52.408,-177.833,5.780,148.375
C08859=1227.993,157.902,-52.387,-177.835,5.778,148.375
C08860=1227.997,157.653,-52.365,-177.838,5.778,148.376
C08861=1228.002,157.404,-52.344,-177.841,5.776,148.376
C08862=1228.007,157.155,-52.322,-177.843,5.775,148.377
C08863=1228.012,156.906,-52.300,-177.846,5.773,148.377
C08864=1228.017,156.656,-52.279,-177.848,5.772,148.378
C08865=1228.022,156.408,-52.257,-177.851,5.771,148.378
C08866=1228.026,156.158,-52.235,-177.853,5.770,148.379
C08867=1228.030,155.910,-52.215,-177.856,5.768,148.379
C08868=1228.035,155.661,-52.193,-177.858,5.767,148.380
C08869=1228.039,155.412,-52.171,-177.861,5.766,148.380
C08870=1228.045,155.162,-52.150,-177.864,5.765,148.381
C08871=1228.049,154.914,-52.128,-177.866,5.764,148.381
C08872=1228.054,154.665,-52.107,-177.868,5.762,148.381
C08873=1228.059,154.415,-52.085,-177.871,5.761,148.382
C08874=1228.063,154.167,-52.064,-177.874,5.760,148.382
C08875=1228.068,153.917,-52.043,-177.876,5.759,148.383
C08876=1228.072,153.668,-52.021,-177.879,5.757,148.383
C08877=1228.077,153.419,-52.000,-177.881,5.756,148.384
C08878=1228.083,153.170,-51.979,-177.884,5.755,148.384
C08879=1228.087,152.922,-51.958,-177.886,5.754,148.385
C08880=1228.091,152.672,-51.936,-177.890,5.752,148.385
C08881=1228.096,152.423,-51.915,-177.892,5.751,148.386
C08882=1228.101,152.174,-51.894,-177.894,5.749,148.386
C08883=1228.106,151.925,-51.872,-177.897,5.749,148.387
C08884=1228.110,151.676,-51.851,-177.899,5.748,148.387
C08885=1228.115,151.427,-51.830,-177.902,5.746,148.388
C08886=1228.120,151.178,-51.809,-177.904,5.745,148.388
C08887=1228.125,150.929,-51.787,-177.907,5.743,148.389
C08888=1228.129,150.680,-51.766,-177.909,5.743,148.389
C08889=1228.134,150.431,-51.744,-177.912,5.741,148.390
C08890=1228.139,150.182,-51.724,-177.915,5.740,148.390
C08891=1228.144,149.932,-51.703,-177.917,5.738,148.391
C08892=1228.148,149.684,-51.681,-177.920,5.738,148.391
C08893=1228.153,149.434,-51.660,-177.922,5.737,148.392
C08894=1228.158,149.185,-51.638,-177.925,5.735,148.392
C08895=1228.162,148.936,-51.618,-177.927,5.734,148.393
C08896=1228.167,148.688,-51.596,-177.930,5.732,148.393
C08897=1228.172,148.439,-51.575,-177.933,5.732,148.394
C08898=1228.176,148.189,-51.555,-177.935,5.730,148.394
C08899=1228.181,147.940,-51.533,-177.938,5.729,148.395
C08900=1228.186,147.691,-51.512,-177.941,5.728,148.395
C08901=1228.190,147.442,-51.492,-177.943,5.727,148.395
C08902=1228.195,147.193,-51.470,-177.945,5.726,148.396
C08903=1228.200,146.944,-51.449,-177.948,5.724,148.396
C08904=1228.204,146.695,-51.428,-177.951,5.723,148.397
C08905=1228.209,146.446,-51.407,-177.953,5.722,148.397
C08906=1228.214,146.197,-51.386,-177.956,5.721,148.398
C08907=1228.219,145.948,-51.365,-177.958,5.719,148.398
C08908=1228.224,145.698,-51.344,-177.961,5.718,148.399
C08909=1228.228,145.450,-51.323,-177.963,5.718,148.399
C08910=1228.233,145.200,-51.302,-177.966,5.716,148.400
C08911=1228.238,144.951,-51.281,-177.968,5.715,148.400
C08912=1228.242,144.702,-51.261,-177.971,5.713,148.401
C08913=1228.247,144.453,-51.239,-177.974,5.713,148.401
C08914=1228.251,144.204,-51.218,-177.976,5.712,148.402
C08915=1228.257,143.955,-51.198,-177.979,5.710,148.402
C08916=1228.261,143.706,-51.177,-177.981,5.709,148.403
C08917=1228.266,143.457,-51.156,-177.984,5.708,148.403
C08918=1228.271,143.208,-51.134,-177.986,5.707,148.404
C08919=1228.275,142.959,-51.114,-177.988,5.706,148.404
C08920=1228.280,142.709,-51.093,-177.992,5.704,148.405
C08921=1228.285,142.460,-51.072,-177.994,5.703,148.405
C08922=1228.290,142.211,-51.051,-177.997,5.702,148.406
C08923=1228.294,141.962,-51.031,-177.999,5.701,148.406
C08924=1228.299,141.713,-51.010,-178.002,5.700,148.407
C08925=1228.303,141.465,-50.989,-178.004,5.698,148.407
C08926=1228.309,141.215,-50.968,-178.007,5.698,148.408
C08927=1228.313,140.966,-50.948,-178.009,5.696,148.408
C08928=1228.318,140.717,-50.927,-178.012,5.695,148.409
C08929=1228.323,140.468,-50.906,-178.014,5.694,148.409
C08930=1228.328,140.219,-50.885,-178.017,5.693,148.410
C08931=1228.332,139.969,-50.865,-178.019,5.692,148.410
C08932=1228.336,139.720,-50.844,-178.023,5.690,148.411
C08933=1228.341,139.471,-50.823,-178.025,5.689,148.411
C08934=1228.346,139.222,-50.803,-178.027,5.688,148.412
C08935=1228.351,138.973,-50.782,-178.030,5.687,148.412
C08936=1228.355,138.724,-50.762,-178.032,5.686,148.413
C08937=1228.361,138.475,-50.741,-178.035,5.685,148.413
C08938=1228.365,138.226,-50.720,-178.037,5.683,148.414
C08939=1228.369,137.977,-50.700,-178.040,5.683,148.414
C08940=1228.375,137.727,-50.679,-178.043,5.681,148.415
C08941=1228.379,137.479,-50.659,-178.045,5.680,148.415
C08942=1228.384,137.229,-50.638,-178.047,5.679,148.416
C08943=1228.389,136.980,-50.617,-178.051,5.678,148.416
C08944=1228.393,136.731,-50.597,-178.053,5.677,148.417
C08945=1228.398,136.482,-50.576,-178.055,5.676,148.417
C08946=1228.403,136.233,-50.555,-178.058,5.674,148.418
C08947=1228.407,135.984,-50.536,-178.061,5.674,148.418
C08948=1228.413,135.734,-50.515,-178.063,5.673,148.419
C08949=1228.417,135.485,-50.494,-178.066,5.671,148.419
C08950=1228.421,135.236,-50.474,-178.068,5.670,148.420
C08951=1228.427,134.987,-50.453,-178.071,5.669,148.420
C08952=1228.431,134.738,-50.433,-178.073,5.668,148.421
C08953=1228.436,134.489,-50.412,-178.076,5.667,148.421
C08954=1228.441,134.239,-50.392,-178.078,5.665,148.422
C08955=1228.446,133.971,-50.370,-178.081,5.665,148.423
C08956=1228.451,133.703,-50.348,-178.084,5.663,148.423
C08957=1228.457,133.434,-50.326,-178.086,5.662,148.424
C08958=1228.462,133.166,-50.304,-178.089,5.661,148.424
C08959=1228.466,132.917,-50.284,-178.092,5.660,148.425
C08960=1228.471,132.667,-50.264,-178.094,5.659,148.425
C08961=1228.476,132.418,-50.243,-178.097,5.658,148.426
C08962=1228.481,132.169,-50.223,-178.099,5.657,148.426
C08963=1228.485,131.920,-50.202,-178.102,5.656,148.427
C08964=1228.490,131.670,-50.182,-178.105,5.654,148.427
C08965=1228.494,131.422,-50.162,-178.107,5.654,148.428
C08966=1228.500,131.172,-50.141,-178.109,5.653,148.428
C08967=1228.504,130.923,-50.121,-178.113,5.651,148.429
C08968=1228.509,130.674,-50.101,-178.115,5.650,148.429
C08969=1228.513,130.425,-50.081,-178.117,5.650,148.430
C08970=1228.519,130.176,-50.061,-178.120,5.648,148.430
C08971=1228.524,129.927,-50.040,-178.123,5.647,148.431
C08972=1228.528,129.678,-50.020,-178.125,5.647,148.432
C08973=1228.533,129.428,-50.000,-178.128,5.645,148.432
C08974=1228.537,129.179,-49.980,-178.131,5.644,148.433
C08975=1228.542,128.930,-49.960,-178.133,5.643,148.433
C08976=1228.547,128.680,-49.939,-178.136,5.642,148.434
C08977=1228.552,128.431,-49.919,-178.138,5.641,148.434
C08978=1228.557,128.183,-49.899,-178.141,5.640,148.435
C08979=1228.561,127.934,-49.879,-178.143,5.638,148.435
C08980=1228.566,127.685,-49.859,-178.146,5.638,148.436
C08981=1228.571,127.435,-49.839,-178.148,5.637,148.436
C08982=1228.575,127.186,-49.819,-178.151,5.635,148.437
C08983=1228.581,126.936,-49.799,-178.153,5.634,148.437
C08984=1228.585,126.687,-49.778,-178.156,5.634,148.438
C08985=1228.590,126.439,-49.758,-178.158,5.633,148.438
C08986=1228.595,126.190,-49.739,-178.161,5.631,148.439
C08987=1228.599,125.941,-49.718,-178.164,5.631,148.439
C08988=1228.604,125.691,-49.699,-178.166,5.630,148.440
C08989=1228.608,125.442,-49.678,-178.169,5.628,148.440
C08990=1228.614,125.193,-49.659,-178.171,5.627,148.441
C08991=1228.618,124.944,-49.639,-178.174,5.627,148.441
C08992=1228.623,124.695,-49.619,-178.176,5.625,148.442
C08993=1228.627,124.446,-49.599,-178.179,5.624,148.442
C08994=1228.632,124.196,-49.579,-178.182,5.623,148.443
C08995=1228.638,123.947,-49.559,-178.184,5.623,148.444
C08996=1228.643,123.698,-49.539,-178.187,5.621,148.444
C08997=1228.647,123.448,-49.519,-178.189,5.620,148.445
C08998=1228.652,123.199,-49.499,-178.192,5.619,148.445
C08999=1228.657,122.950,-49.479,-178.194,5.618,148.446
C09000=1228.662,122.702,-49.459,-178.197,5.617,148.446
C09001=1228.666,122.452,-49.439,-178.199,5.616,148.447
C09002=1228.671,122.203,-49.420,-178.202,5.615,148.447
C09003=1228.675,121.954,-49.399,-178.205,5.614,148.448
C09004=1228.681,121.705,-49.380,-178.207,5.613,148.448
C09005=1228.686,121.455,-49.360,-178.209,5.612,148.449
C09006=1228.690,121.206,-49.340,-178.212,5.611,148.449
C09007=1228.695,120.957,-49.320,-178.215,5.610,148.450
C09008=1228.700,120.708,-49.301,-178.217,5.609,148.451
C09009=1228.705,120.459,-49.281,-178.219,5.608,148.451
C09010=1228.709,120.210,-49.262,-178.223,5.607,148.452
C09011=1228.713,119.960,-49.242,-178.225,5.606,148.452
C09012=1228.718,119.712,-49.222,-178.227,5.605,148.453
C09013=1228.723,119.462,-49.202,-178.230,5.605,148.453
C09014=1228.728,119.213,-49.183,-178.233,5.603,148.454
C09015=1228.733,118.964,-49.163,-178.235,5.602,148.454
C09016=1228.738,118.715,-49.143,-178.237,5.601,148.455
C09017=1228.742,118.465,-49.123,-178.241,5.600,148.455
C09018=1228.747,118.216,-49.104,-178.243,5.599,148.456
C09019=1228.752,117.967,-49.084,-178.245,5.598,148.456
C09020=1228.757,117.718,-49.064,-178.248,5.598,148.457
C09021=1228.762,117.468,-49.044,-178.251,5.596,148.457
C09022=1228.766,117.220,-49.026,-178.253,5.595,148.458
C09023=1228.771,116.970,-49.006,-178.255,5.594,148.458
C09024=1228.776,116.721,-48.986,-178.258,5.594,148.459
C09025=1228.781,116.472,-48.966,-178.261,5.592,148.460
C09026=1228.785,116.223,-48.947,-178.263,5.591,148.460
C09027=1228.790,115.973,-48.927,-178.266,5.590,148.461
C09028=1228.796,115.724,-48.908,-178.268,5.590,148.461
C09029=1228.800,115.475,-48.889,-178.271,5.588,148.462
C09030=1228.804,115.226,-48.869,-178.274,5.587,148.462
C09031=1228.810,114.977,-48.850,-178.276,5.586,148.463
C09032=1228.814,114.727,-48.830,-178.278,5.586,148.464
C09033=1228.819,114.479,-48.810,-178.282,5.584,148.464
C09034=1228.823,114.230,-48.791,-178.284,5.583,148.465
C09035=1228.828,113.980,-48.771,-178.286,5.583,148.465
C09036=1228.834,113.731,-48.752,-178.288,5.582,148.466
C09037=1228.838,113.482,-48.732,-178.291,5.581,148.466
C09038=1228.843,113.232,-48.713,-178.294,5.580,148.467
C09039=1228.848,112.983,-48.694,-178.296,5.579,148.467
C09040=1228.852,112.734,-48.674,-178.299,5.578,148.468
C09041=1228.858,112.485,-48.655,-178.302,5.578,148.469
C09042=1228.862,112.235,-48.635,-178.304,5.576,148.469
C09043=1228.866,111.986,-48.616,-178.307,5.575,148.470
C09044=1228.872,111.737,-48.597,-178.309,5.574,148.470
C09045=1228.877,111.488,-48.577,-178.312,5.574,148.471
C09046=1228.882,111.239,-48.558,-178.314,5.573,148.471
C09047=1228.886,110.990,-48.539,-178.317,5.571,148.472
C09048=1228.891,110.740,-48.519,-178.320,5.571,148.472
C09049=1228.896,110.491,-48.500,-178.322,5.570,148.473
C09050=1228.900,110.242,-48.481,-178.324,5.569,148.473
C09051=1228.905,109.993,-48.462,-178.327,5.567,148.474
C09052=1228.910,109.743,-48.442,-178.330,5.567,148.474
C09053=1228.915,109.495,-48.423,-178.332,5.566,148.475
C09054=1228.920,109.245,-48.405,-178.335,5.565,148.476
C09055=1228.925,108.996,-48.385,-178.337,5.564,148.476
C09056=1228.929,108.747,-48.366,-178.340,5.563,148.477
C09057=1228.934,108.497,-48.347,-178.343,5.562,148.477
C09058=1228.939,108.248,-48.327,-178.345,5.561,148.478
C09059=1228.944,107.980,-48.306,-178.347,5.561,148.478
C09060=1228.950,107.711,-48.286,-178.351,5.559,148.479
C09061=1228.954,107.443,-48.266,-178.353,5.559,148.480
C09062=1228.960,107.175,-48.245,-178.356,5.557,148.480
C09063=1228.964,106.925,-48.225,-178.359,5.556,148.481
C09064=1228.969,106.677,-48.207,-178.361,5.556,148.481
C09065=1228.974,106.426,-48.188,-178.364,5.555,148.482
C09066=1228.979,106.178,-48.168,-178.366,5.554,148.483
C09067=1228.983,105.928,-48.149,-178.369,5.553,148.483
C09068=1228.989,105.679,-48.130,-178.372,5.552,148.484
C09069=1228.993,105.430,-48.112,-178.374,5.551,148.484
C09070=1228.998,105.181,-48.092,-178.376,5.550,148.485
C09071=1229.003,104.931,-48.073,-178.379,5.550,148.485
C09072=1229.008,104.683,-48.054,-178.381,5.549,148.486
C09073=1229.013,104.432,-48.035,-178.384,5.547,148.487
C09074=1229.017,104.184,-48.016,-178.387,5.547,148.487
C09075=1229.022,103.934,-47.997,-178.389,5.546,148.488
C09076=1229.027,103.686,-47.978,-178.392,5.545,148.488
C09077=1229.032,103.435,-47.959,-178.394,5.545,148.489
C09078=1229.036,103.187,-47.940,-178.396,5.544,148.489
C09079=1229.041,102.937,-47.921,-178.400,5.542,148.490
C09080=1229.046,102.688,-47.903,-178.402,5.542,148.491
C09081=1229.051,102.439,-47.883,-178.404,5.541,148.491
C09082=1229.055,102.190,-47.864,-178.407,5.540,148.492
C09083=1229.061,101.941,-47.846,-178.410,5.539,148.492
C09084=1229.065,101.691,-47.827,-178.412,5.538,148.493
C09085=1229.070,101.442,-47.807,-178.415,5.537,148.493
C09086=1229.075,101.193,-47.789,-178.418,5.536,148.494
C09087=1229.080,100.944,-47.770,-178.420,5.535,148.494
C09088=1229.085,100.695,-47.752,-178.422,5.535,148.495
C09089=1229.090,100.445,-47.732,-178.425,5.534,148.496
C09090=1229.094,100.196,-47.714,-178.427,5.533,148.496
C09091=1229.099,99.946,-47.695,-178.430,5.532,148.497
C09092=1229.104,99.698,-47.676,-178.433,5.531,148.497
C09093=1229.109,99.448,-47.658,-178.435,5.531,148.498
C09094=1229.114,99.199,-47.638,-178.438,5.530,148.498
C09095=1229.118,98.950,-47.620,-178.440,5.529,148.499
C09096=1229.123,98.700,-47.601,-178.443,5.528,148.500
C09097=1229.128,98.451,-47.583,-178.445,5.527,148.500
C09098=1229.133,98.202,-47.563,-178.448,5.526,148.501
C09099=1229.138,97.952,-47.545,-178.451,5.525,148.501
C09100=1229.142,97.704,-47.526,-178.453,5.524,148.502
C09101=1229.147,97.453,-47.507,-178.455,5.524,148.503
C09102=1229.152,97.205,-47.489,-178.458,5.523,148.503
C09103=1229.157,96.956,-47.471,-178.460,5.522,148.504
C09104=1229.162,96.706,-47.451,-178.463,5.521,148.504
C09105=1229.167,96.457,-47.433,-178.466,5.520,148.505
C09106=1229.172,96.208,-47.414,-178.469,5.520,148.506
C09107=1229.176,95.958,-47.395,-178.471,5.519,148.506
C09108=1229.181,95.709,-47.377,-178.473,5.518,148.507
C09109=1229.187,95.460,-47.358,-178.476,5.517,148.507
C09110=1229.191,95.210,-47.340,-178.478,5.516,148.508
C09111=1229.195,94.962,-47.321,-178.481,5.515,148.508
C09112=1229.201,94.712,-47.303,-178.484,5.514,148.509
C09113=1229.205,94.462,-47.284,-178.487,5.514,148.510
C09114=1229.210,94.214,-47.265,-178.489,5.513,148.510
C09115=1229.215,93.965,-47.248,-178.491,5.512,148.511
C09116=1229.220,93.714,-47.229,-178.494,5.512,148.511
C09117=1229.225,93.466,-47.210,-178.496,5.511,148.512
C09118=1229.229,93.217,-47.192,-178.499,5.510,148.512
C09119=1229.235,92.967,-47.173,-178.502,5.509,148.513
C09120=1229.239,92.718,-47.154,-178.504,5.508,148.514
C09121=1229.244,92.469,-47.136,-178.507,5.507,148.514
C09122=1229.249,92.220,-47.118,-178.509,5.506,148.515
C09123=1229.254,91.970,-47.099,-178.512,5.506,148.515
C09124=1229.259,91.721,-47.081,-178.514,5.505,148.516
C09125=1229.264,91.472,-47.063,-178.517,5.504,148.517
C09126=1229.268,91.223,-47.045,-178.519,5.504,148.517
C09127=1229.272,90.973,-47.026,-178.522,5.502,148.518
